KUKA KRL data list: Fadenlegen.dat

&ACCESS RVP
&REL 24
&PARAM DISKPATH = KRC:\R1\myProgramme\Mahlen
DEFDAT  Fadenlegen
;FOLD EXTERNAL DECLARATIONS;%{PE}%MKUKATPBASIS,%CEXT,%VCOMMON,%P
;FOLD BASISTECH EXT;%{PE}%MKUKATPBASIS,%CEXT,%VEXT,%P
EXT  BAS (BAS_COMMAND  :IN,REAL  :IN )
;ENDFOLD (BASISTECH EXT)
;FOLD USER EXT;%{E}%MKUKATPUSER,%CEXT,%VEXT,%P
;Make your modifications here

DECL E6POS KM={X 270.508820,Y 129.418152,Z 50.0000,A 0.0,B -180.000,C 0.0,S 6,T 26,E1 0.0,E2 0.0,E3 0.0,E4 0.0,E5 0.0,E6 0.0}

DECL E6POS test1={X 276.364288,Y 142.737,Z 19.5319443,A 180.000,B -180.000,C 0.0,S 2,T 10,E1 0.0,E2 0.0,E3 0.0,E4 0.0,E5 0.0,E6 0.0}

DECL E6AXIS MyHome={A1 4.82899427,A2 -40.7993927,A3 107.255463,A4 -2.92958689,A5 26.5940895,A6 -79.3028717,E1 0.0,E2 0.0,E3 0.0,E4 0.0,E5 0.0,E6 0.0}

DECL INT turn=1

DECL INT LetztePos
DECL INT len_Punkte=4002; 4002

DECL INT Sturz[180]
Sturz[1]=10
Sturz[2]=10
Sturz[3]=10
Sturz[4]=10
Sturz[5]=10
Sturz[6]=10
Sturz[7]=10
Sturz[8]=10
Sturz[9]=10
Sturz[10]=10
Sturz[11]=10
Sturz[12]=10
Sturz[13]=10
Sturz[14]=10
Sturz[15]=10
Sturz[16]=10
Sturz[17]=10
Sturz[18]=10
Sturz[19]=10
Sturz[20]=10
Sturz[21]=10
Sturz[22]=10
Sturz[23]=10
Sturz[24]=10
Sturz[25]=10
Sturz[26]=10
Sturz[27]=10
Sturz[28]=10
Sturz[29]=10
Sturz[30]=10
Sturz[31]=10
Sturz[32]=10
Sturz[33]=10
Sturz[34]=10
Sturz[35]=10
Sturz[36]=10
Sturz[37]=10
Sturz[38]=10
Sturz[39]=10
Sturz[40]=10
Sturz[41]=10
Sturz[42]=10
Sturz[43]=10
Sturz[44]=10
Sturz[45]=10
Sturz[46]=10
Sturz[47]=10
Sturz[48]=10
Sturz[49]=10
Sturz[50]=10
Sturz[51]=10
Sturz[52]=10
Sturz[53]=10
Sturz[54]=10
Sturz[55]=10
Sturz[56]=10
Sturz[57]=10
Sturz[58]=10
Sturz[59]=10
Sturz[60]=10
Sturz[61]=10
Sturz[62]=10
Sturz[63]=10
Sturz[64]=10
Sturz[65]=10
Sturz[66]=10
Sturz[67]=10
Sturz[68]=10
Sturz[69]=10
Sturz[70]=10
Sturz[71]=10
Sturz[72]=10
Sturz[73]=10
Sturz[74]=10
Sturz[75]=10
Sturz[76]=10
Sturz[77]=10
Sturz[78]=10
Sturz[79]=10
Sturz[80]=10
Sturz[81]=10
Sturz[82]=10
Sturz[83]=10
Sturz[84]=10
Sturz[85]=10
Sturz[86]=10
Sturz[87]=10
Sturz[88]=10
Sturz[89]=10
Sturz[90]=10
Sturz[91]=-10
Sturz[92]=-10
Sturz[93]=-10
Sturz[94]=-10
Sturz[95]=-10
Sturz[96]=-10
Sturz[97]=-10
Sturz[98]=-10
Sturz[99]=-10
Sturz[100]=-10
Sturz[101]=-10
Sturz[102]=-10
Sturz[103]=-10
Sturz[104]=-10
Sturz[105]=-10
Sturz[106]=-10
Sturz[107]=-10
Sturz[108]=-10
Sturz[109]=-10
Sturz[110]=-10
Sturz[111]=-10
Sturz[112]=10
Sturz[113]=10
Sturz[114]=10
Sturz[115]=10
Sturz[116]=10
Sturz[117]=10
Sturz[118]=10
Sturz[119]=10
Sturz[120]=10
Sturz[121]=10
Sturz[122]=10
Sturz[123]=10
Sturz[124]=10
Sturz[125]=10
Sturz[126]=10
Sturz[127]=10
Sturz[128]=10
Sturz[129]=10
Sturz[130]=10
Sturz[131]=10
Sturz[132]=10
Sturz[133]=10
Sturz[134]=10
Sturz[135]=10
Sturz[136]=10
Sturz[137]=10
Sturz[138]=10
Sturz[139]=10
Sturz[140]=10
Sturz[141]=10
Sturz[142]=10
Sturz[143]=10
Sturz[144]=10
Sturz[145]=10
Sturz[146]=10
Sturz[147]=10
Sturz[148]=10
Sturz[149]=10
Sturz[150]=10
Sturz[151]=10
Sturz[152]=10
Sturz[153]=10
Sturz[154]=10
Sturz[155]=10
Sturz[156]=10
Sturz[157]=10
Sturz[158]=10
Sturz[159]=10
Sturz[160]=10
Sturz[161]=10
Sturz[162]=10
Sturz[163]=10
Sturz[164]=10
Sturz[165]=10
Sturz[166]=10
Sturz[167]=10
Sturz[168]=10
Sturz[169]=10
Sturz[170]=10
Sturz[171]=10
Sturz[172]=10
Sturz[173]=10
Sturz[174]=10
Sturz[175]=10
Sturz[176]=10
Sturz[177]=10
Sturz[178]=10
Sturz[179]=10
Sturz[180]=10



DECL INT TEST[374]
TEST[1]=0
TEST[2]=22
TEST[3]=1
TEST[4]=23
TEST[5]=2
TEST[6]=24
TEST[7]=3
TEST[8]=25
TEST[9]=4
TEST[10]=26
TEST[11]=5
TEST[12]=27
TEST[13]=6
TEST[14]=28
TEST[15]=7
TEST[16]=29
TEST[17]=8
TEST[18]=30
TEST[19]=9
TEST[20]=31
TEST[21]=10
TEST[22]=32
TEST[23]=11
TEST[24]=33
TEST[25]=12
TEST[26]=34
TEST[27]=13
TEST[28]=35
TEST[29]=14
TEST[30]=36
TEST[31]=15
TEST[32]=37
TEST[33]=16
TEST[34]=38
TEST[35]=17
TEST[36]=39
TEST[37]=18
TEST[38]=40
TEST[39]=19
TEST[40]=41
TEST[41]=20
TEST[42]=42
TEST[43]=21
TEST[44]=43
TEST[45]=22
TEST[46]=44
TEST[47]=23
TEST[48]=45
TEST[49]=24
TEST[50]=46
TEST[51]=25
TEST[52]=47
TEST[53]=26
TEST[54]=48
TEST[55]=27
TEST[56]=49
TEST[57]=28
TEST[58]=50
TEST[59]=29
TEST[60]=51
TEST[61]=30
TEST[62]=52
TEST[63]=31
TEST[64]=53
TEST[65]=32
TEST[66]=54
TEST[67]=33
TEST[68]=55
TEST[69]=34
TEST[70]=56
TEST[71]=35
TEST[72]=57
TEST[73]=36
TEST[74]=58
TEST[75]=37
TEST[76]=59
TEST[77]=38
TEST[78]=60
TEST[79]=39
TEST[80]=61
TEST[81]=40
TEST[82]=62
TEST[83]=41
TEST[84]=63
TEST[85]=42
TEST[86]=64
TEST[87]=43
TEST[88]=65
TEST[89]=44
TEST[90]=66
TEST[91]=45
TEST[92]=67
TEST[93]=46
TEST[94]=68
TEST[95]=47
TEST[96]=69
TEST[97]=48
TEST[98]=70
TEST[99]=49
TEST[100]=71
TEST[101]=50
TEST[102]=72
TEST[103]=51
TEST[104]=73
TEST[105]=52
TEST[106]=74
TEST[107]=53
TEST[108]=75
TEST[109]=54
TEST[110]=76
TEST[111]=55
TEST[112]=77
TEST[113]=56
TEST[114]=78
TEST[115]=57
TEST[116]=79
TEST[117]=58
TEST[118]=80
TEST[119]=59
TEST[120]=81
TEST[121]=60
TEST[122]=82
TEST[123]=61
TEST[124]=83
TEST[125]=62
TEST[126]=84
TEST[127]=63
TEST[128]=85
TEST[129]=64
TEST[130]=86
TEST[131]=65
TEST[132]=87
TEST[133]=66
TEST[134]=88
TEST[135]=67
TEST[136]=89
TEST[137]=68
TEST[138]=90
TEST[139]=69
TEST[140]=91
TEST[141]=70
TEST[142]=92
TEST[143]=71
TEST[144]=93
TEST[145]=72
TEST[146]=94
TEST[147]=73
TEST[148]=95
TEST[149]=74
TEST[150]=96
TEST[151]=75
TEST[152]=97
TEST[153]=76
TEST[154]=98
TEST[155]=77
TEST[156]=99
TEST[157]=78
TEST[158]=100
TEST[159]=79
TEST[160]=101
TEST[161]=80
TEST[162]=102
TEST[163]=81
TEST[164]=103
TEST[165]=82
TEST[166]=104
TEST[167]=83
TEST[168]=105
TEST[169]=84
TEST[170]=106
TEST[171]=85
TEST[172]=107
TEST[173]=86
TEST[174]=108
TEST[175]=87
TEST[176]=109
TEST[177]=88
TEST[178]=110
TEST[179]=89
TEST[180]=111
TEST[181]=90
TEST[182]=112
TEST[183]=91
TEST[184]=113
TEST[185]=92
TEST[186]=114
TEST[187]=93
TEST[188]=115
TEST[189]=94
TEST[190]=116
TEST[191]=95
TEST[192]=117
TEST[193]=96
TEST[194]=118
TEST[195]=97
TEST[196]=119
TEST[197]=98
TEST[198]=120
TEST[199]=99
TEST[200]=121
TEST[201]=100
TEST[202]=122
TEST[203]=101
TEST[204]=123
TEST[205]=102
TEST[206]=124
TEST[207]=103
TEST[208]=125
TEST[209]=104
TEST[210]=126
TEST[211]=105
TEST[212]=127
TEST[213]=106
TEST[214]=128
TEST[215]=107
TEST[216]=129
TEST[217]=108
TEST[218]=130
TEST[219]=109
TEST[220]=131
TEST[221]=110
TEST[222]=132
TEST[223]=111
TEST[224]=133
TEST[225]=112
TEST[226]=134
TEST[227]=113
TEST[228]=135
TEST[229]=114
TEST[230]=136
TEST[231]=115
TEST[232]=137
TEST[233]=116
TEST[234]=138
TEST[235]=117
TEST[236]=139
TEST[237]=118
TEST[238]=140
TEST[239]=119
TEST[240]=141
TEST[241]=120
TEST[242]=142
TEST[243]=121
TEST[244]=143
TEST[245]=122
TEST[246]=144
TEST[247]=123
TEST[248]=145
TEST[249]=124
TEST[250]=146
TEST[251]=125
TEST[252]=147
TEST[253]=126
TEST[254]=148
TEST[255]=127
TEST[256]=149
TEST[257]=128
TEST[258]=150
TEST[259]=129
TEST[260]=151
TEST[261]=130
TEST[262]=152
TEST[263]=131
TEST[264]=153
TEST[265]=132
TEST[266]=154
TEST[267]=133
TEST[268]=155
TEST[269]=134
TEST[270]=156
TEST[271]=135
TEST[272]=157
TEST[273]=136
TEST[274]=158
TEST[275]=137
TEST[276]=159
TEST[277]=138
TEST[278]=160
TEST[279]=139
TEST[280]=161
TEST[281]=140
TEST[282]=162
TEST[283]=141
TEST[284]=163
TEST[285]=142
TEST[286]=164
TEST[287]=143
TEST[288]=165
TEST[289]=144
TEST[290]=166
TEST[291]=145
TEST[292]=167
TEST[293]=146
TEST[294]=168
TEST[295]=147
TEST[296]=169
TEST[297]=148
TEST[298]=170
TEST[299]=149
TEST[300]=171
TEST[301]=150
TEST[302]=172
TEST[303]=151
TEST[304]=173
TEST[305]=152
TEST[306]=174
TEST[307]=153
TEST[308]=175
TEST[309]=154
TEST[310]=176
TEST[311]=155
TEST[312]=177
TEST[313]=156
TEST[314]=178
TEST[315]=157
TEST[316]=179
TEST[317]=158
TEST[318]=1
TEST[319]=159
TEST[320]=2
TEST[321]=160
TEST[322]=3
TEST[323]=161
TEST[324]=4
TEST[325]=162
TEST[326]=5
TEST[327]=163
TEST[328]=6
TEST[329]=164
TEST[330]=7
TEST[331]=165
TEST[332]=8
TEST[333]=166
TEST[334]=9
TEST[335]=167
TEST[336]=10
TEST[337]=168
TEST[338]=11
TEST[339]=169
TEST[340]=12
TEST[341]=170
TEST[342]=13
TEST[343]=171
TEST[344]=14
TEST[345]=172
TEST[346]=15
TEST[347]=173
TEST[348]=16
TEST[349]=174
TEST[350]=17
TEST[351]=175
TEST[352]=18
TEST[353]=176
TEST[354]=19
TEST[355]=177
TEST[356]=20
TEST[357]=178
TEST[358]=21
TEST[359]=179
TEST[360]=22
TEST[361]=1
TEST[362]=23
TEST[363]=2
TEST[364]=24
TEST[365]=3
TEST[366]=25
TEST[367]=4
TEST[368]=26
TEST[369]=5
TEST[370]=27
TEST[371]=6
TEST[372]=28
TEST[373]=7
TEST[374]=29





DECL INT Punkte[4002]
Punkte[1]=0
Punkte[2]=98
Punkte[3]=1
Punkte[4]=99
Punkte[5]=4
Punkte[6]=76
Punkte[7]=7
Punkte[8]=93
Punkte[9]=169
Punkte[10]=86
Punkte[11]=13
Punkte[12]=123
Punkte[13]=14
Punkte[14]=87
Punkte[15]=170
Punkte[16]=95
Punkte[17]=8
Punkte[18]=77
Punkte[19]=9
Punkte[20]=79
Punkte[21]=161
Punkte[22]=78
Punkte[23]=11
Punkte[24]=109
Punkte[25]=10
Punkte[26]=108
Punkte[27]=43
Punkte[28]=152
Punkte[29]=67
Punkte[30]=144
Punkte[31]=65
Punkte[32]=143
Punkte[33]=64
Punkte[34]=137
Punkte[35]=33
Punkte[36]=99
Punkte[37]=176
Punkte[38]=88
Punkte[39]=163
Punkte[40]=80
Punkte[41]=12
Punkte[42]=81
Punkte[43]=174
Punkte[44]=103
Punkte[45]=5
Punkte[46]=85
Punkte[47]=13
Punkte[48]=112
Punkte[49]=37
Punkte[50]=140
Punkte[51]=58
Punkte[52]=131
Punkte[53]=20
Punkte[54]=120
Punkte[55]=6
Punkte[56]=104
Punkte[57]=179
Punkte[58]=89
Punkte[59]=178
Punkte[60]=75
Punkte[61]=156
Punkte[62]=53
Punkte[63]=168
Punkte[64]=79
Punkte[65]=11
Punkte[66]=78
Punkte[67]=10
Punkte[68]=122
Punkte[69]=9
Punkte[70]=77
Punkte[71]=158
Punkte[72]=84
Punkte[73]=167
Punkte[74]=85
Punkte[75]=4
Punkte[76]=102
Punkte[77]=6
Punkte[78]=91
Punkte[79]=7
Punkte[80]=76
Punkte[81]=157
Punkte[82]=54
Punkte[83]=129
Punkte[84]=53
Punkte[85]=166
Punkte[86]=83
Punkte[87]=165
Punkte[88]=101
Punkte[89]=3
Punkte[90]=98
Punkte[91]=173
Punkte[92]=78
Punkte[93]=160
Punkte[94]=81
Punkte[95]=12
Punkte[96]=80
Punkte[97]=10
Punkte[98]=85
Punkte[99]=168
Punkte[100]=92
Punkte[101]=7
Punkte[102]=121
Punkte[103]=13
Punkte[104]=82
Punkte[105]=148
Punkte[106]=76
Punkte[107]=146
Punkte[108]=75
Punkte[109]=2
Punkte[110]=100
Punkte[111]=4
Punkte[112]=79
Punkte[113]=8
Punkte[114]=106
Punkte[115]=6
Punkte[116]=77
Punkte[117]=9
Punkte[118]=107
Punkte[119]=42
Punkte[120]=151
Punkte[121]=74
Punkte[122]=145
Punkte[123]=73
Punkte[124]=144
Punkte[125]=64
Punkte[126]=143
Punkte[127]=12
Punkte[128]=111
Punkte[129]=36
Punkte[130]=127
Punkte[131]=28
Punkte[132]=126
Punkte[133]=26
Punkte[134]=117
Punkte[135]=14
Punkte[136]=84
Punkte[137]=169
Punkte[138]=87
Punkte[139]=10
Punkte[140]=78
Punkte[141]=159
Punkte[142]=77
Punkte[143]=9
Punkte[144]=79
Punkte[145]=11
Punkte[146]=110
Punkte[147]=8
Punkte[148]=96
Punkte[149]=165
Punkte[150]=101
Punkte[151]=166
Punkte[152]=100
Punkte[153]=36
Punkte[154]=140
Punkte[155]=71
Punkte[156]=154
Punkte[157]=72
Punkte[158]=155
Punkte[159]=52
Punkte[160]=167
Punkte[161]=91
Punkte[162]=17
Punkte[163]=124
Punkte[164]=15
Punkte[165]=123
Punkte[166]=12
Punkte[167]=82
Punkte[168]=177
Punkte[169]=80
Punkte[170]=162
Punkte[171]=84
Punkte[172]=3
Punkte[173]=76
Punkte[174]=157
Punkte[175]=77
Punkte[176]=8
Punkte[177]=78
Punkte[178]=164
Punkte[179]=81
Punkte[180]=174
Punkte[181]=87
Punkte[182]=163
Punkte[183]=49
Punkte[184]=119
Punkte[185]=19
Punkte[186]=124
Punkte[187]=16
Punkte[188]=90
Punkte[189]=179
Punkte[190]=73
Punkte[191]=1
Punkte[192]=79
Punkte[193]=10
Punkte[194]=86
Punkte[195]=14
Punkte[196]=111
Punkte[197]=11
Punkte[198]=77
Punkte[199]=146
Punkte[200]=74
Punkte[201]=118
Punkte[202]=48
Punkte[203]=162
Punkte[204]=82
Punkte[205]=148
Punkte[206]=83
Punkte[207]=3
Punkte[208]=99
Punkte[209]=9
Punkte[210]=80
Punkte[211]=12
Punkte[212]=81
Punkte[213]=175
Punkte[214]=98
Punkte[215]=170
Punkte[216]=102
Punkte[217]=168
Punkte[218]=84
Punkte[219]=5
Punkte[220]=75
Punkte[221]=6
Punkte[222]=79
Punkte[223]=147
Punkte[224]=74
Punkte[225]=1
Punkte[226]=94
Punkte[227]=169
Punkte[228]=56
Punkte[229]=139
Punkte[230]=70
Punkte[231]=153
Punkte[232]=78
Punkte[233]=11
Punkte[234]=105
Punkte[235]=3
Punkte[236]=97
Punkte[237]=172
Punkte[238]=96
Punkte[239]=2
Punkte[240]=103
Punkte[241]=39
Punkte[242]=104
Punkte[243]=178
Punkte[244]=72
Punkte[245]=177
Punkte[246]=102
Punkte[247]=171
Punkte[248]=80
Punkte[249]=147
Punkte[250]=75
Punkte[251]=155
Punkte[252]=74
Punkte[253]=118
Punkte[254]=11
Punkte[255]=77
Punkte[256]=10
Punkte[257]=81
Punkte[258]=163
Punkte[259]=93
Punkte[260]=7
Punkte[261]=78
Punkte[262]=12
Punkte[263]=110
Punkte[264]=35
Punkte[265]=100
Punkte[266]=36
Punkte[267]=102
Punkte[268]=5
Punkte[269]=101
Punkte[270]=4
Punkte[271]=112
Punkte[272]=13
Punkte[273]=120
Punkte[274]=21
Punkte[275]=122
Punkte[276]=11
Punkte[277]=109
Punkte[278]=34
Punkte[279]=139
Punkte[280]=87
Punkte[281]=15
Punkte[282]=124
Punkte[283]=14
Punkte[284]=123
Punkte[285]=12
Punkte[286]=142
Punkte[287]=72
Punkte[288]=144
Punkte[289]=66
Punkte[290]=131
Punkte[291]=20
Punkte[292]=97
Punkte[293]=165
Punkte[294]=101
Punkte[295]=166
Punkte[296]=82
Punkte[297]=13
Punkte[298]=85
Punkte[299]=159
Punkte[300]=46
Punkte[301]=115
Punkte[302]=10
Punkte[303]=122
Punkte[304]=9
Punkte[305]=77
Punkte[306]=127
Punkte[307]=36
Punkte[308]=111
Punkte[309]=12
Punkte[310]=116
Punkte[311]=11
Punkte[312]=80
Punkte[313]=4
Punkte[314]=86
Punkte[315]=173
Punkte[316]=96
Punkte[317]=8
Punkte[318]=79
Punkte[319]=3
Punkte[320]=108
Punkte[321]=2
Punkte[322]=84
Punkte[323]=166
Punkte[324]=83
Punkte[325]=5
Punkte[326]=77
Punkte[327]=7
Punkte[328]=76
Punkte[329]=149
Punkte[330]=85
Punkte[331]=160
Punkte[332]=89
Punkte[333]=179
Punkte[334]=75
Punkte[335]=146
Punkte[336]=82
Punkte[337]=11
Punkte[338]=104
Punkte[339]=172
Punkte[340]=98
Punkte[341]=29
Punkte[342]=126
Punkte[343]=17
Punkte[344]=152
Punkte[345]=16
Punkte[346]=125
Punkte[347]=23
Punkte[348]=123
Punkte[349]=13
Punkte[350]=84
Punkte[351]=12
Punkte[352]=80
Punkte[353]=174
Punkte[354]=81
Punkte[355]=175
Punkte[356]=100
Punkte[357]=168
Punkte[358]=53
Punkte[359]=156
Punkte[360]=77
Punkte[361]=8
Punkte[362]=95
Punkte[363]=169
Punkte[364]=85
Punkte[365]=171
Punkte[366]=101
Punkte[367]=167
Punkte[368]=83
Punkte[369]=4
Punkte[370]=99
Punkte[371]=32
Punkte[372]=138
Punkte[373]=69
Punkte[374]=153
Punkte[375]=18
Punkte[376]=124
Punkte[377]=13
Punkte[378]=111
Punkte[379]=45
Punkte[380]=158
Punkte[381]=78
Punkte[382]=12
Punkte[383]=81
Punkte[384]=11
Punkte[385]=77
Punkte[386]=127
Punkte[387]=17
Punkte[388]=125
Punkte[389]=24
Punkte[390]=116
Punkte[391]=47
Punkte[392]=161
Punkte[393]=79
Punkte[394]=7
Punkte[395]=102
Punkte[396]=167
Punkte[397]=86
Punkte[398]=6
Punkte[399]=121
Punkte[400]=8
Punkte[401]=84
Punkte[402]=10
Punkte[403]=136
Punkte[404]=50
Punkte[405]=165
Punkte[406]=78
Punkte[407]=176
Punkte[408]=77
Punkte[409]=128
Punkte[410]=0
Punkte[411]=93
Punkte[412]=164
Punkte[413]=82
Punkte[414]=148
Punkte[415]=14
Punkte[416]=87
Punkte[417]=150
Punkte[418]=15
Punkte[419]=151
Punkte[420]=89
Punkte[421]=178
Punkte[422]=103
Punkte[423]=10
Punkte[424]=88
Punkte[425]=141
Punkte[426]=60
Punkte[427]=170
Punkte[428]=94
Punkte[429]=7
Punkte[430]=121
Punkte[431]=75
Punkte[432]=3
Punkte[433]=101
Punkte[434]=11
Punkte[435]=78
Punkte[436]=172
Punkte[437]=80
Punkte[438]=12
Punkte[439]=79
Punkte[440]=5
Punkte[441]=76
Punkte[442]=157
Punkte[443]=54
Punkte[444]=168
Punkte[445]=97
Punkte[446]=2
Punkte[447]=132
Punkte[448]=29
Punkte[449]=127
Punkte[450]=77
Punkte[451]=161
Punkte[452]=91
Punkte[453]=7
Punkte[454]=105
Punkte[455]=167
Punkte[456]=99
Punkte[457]=33
Punkte[458]=101
Punkte[459]=165
Punkte[460]=51
Punkte[461]=154
Punkte[462]=44
Punkte[463]=109
Punkte[464]=4
Punkte[465]=84
Punkte[466]=159
Punkte[467]=86
Punkte[468]=169
Punkte[469]=57
Punkte[470]=160
Punkte[471]=78
Punkte[472]=10
Punkte[473]=82
Punkte[474]=12
Punkte[475]=142
Punkte[476]=55
Punkte[477]=158
Punkte[478]=83
Punkte[479]=11
Punkte[480]=92
Punkte[481]=0
Punkte[482]=128
Punkte[483]=38
Punkte[484]=103
Punkte[485]=174
Punkte[486]=81
Punkte[487]=157
Punkte[488]=47
Punkte[489]=164
Punkte[490]=99
Punkte[491]=175
Punkte[492]=91
Punkte[493]=6
Punkte[494]=76
Punkte[495]=7
Punkte[496]=84
Punkte[497]=134
Punkte[498]=85
Punkte[499]=140
Punkte[500]=52
Punkte[501]=155
Punkte[502]=45
Punkte[503]=158
Punkte[504]=48
Punkte[505]=118
Punkte[506]=74
Punkte[507]=145
Punkte[508]=75
Punkte[509]=156
Punkte[510]=53
Punkte[511]=166
Punkte[512]=90
Punkte[513]=0
Punkte[514]=128
Punkte[515]=18
Punkte[516]=125
Punkte[517]=25
Punkte[518]=126
Punkte[519]=31
Punkte[520]=133
Punkte[521]=79
Punkte[522]=11
Punkte[523]=119
Punkte[524]=12
Punkte[525]=78
Punkte[526]=168
Punkte[527]=60
Punkte[528]=170
Punkte[529]=59
Punkte[530]=141
Punkte[531]=88
Punkte[532]=150
Punkte[533]=15
Punkte[534]=151
Punkte[535]=16
Punkte[536]=91
Punkte[537]=166
Punkte[538]=101
Punkte[539]=37
Punkte[540]=112
Punkte[541]=13
Punkte[542]=123
Punkte[543]=14
Punkte[544]=93
Punkte[545]=171
Punkte[546]=62
Punkte[547]=142
Punkte[548]=63
Punkte[549]=143
Punkte[550]=12
Punkte[551]=83
Punkte[552]=165
Punkte[553]=96
Punkte[554]=164
Punkte[555]=88
Punkte[556]=140
Punkte[557]=52
Punkte[558]=166
Punkte[559]=102
Punkte[560]=37
Punkte[561]=112
Punkte[562]=177
Punkte[563]=94
Punkte[564]=0
Punkte[565]=128
Punkte[566]=179
Punkte[567]=77
Punkte[568]=153
Punkte[569]=70
Punkte[570]=145
Punkte[571]=69
Punkte[572]=171
Punkte[573]=98
Punkte[574]=1
Punkte[575]=130
Punkte[576]=55
Punkte[577]=169
Punkte[578]=56
Punkte[579]=159
Punkte[580]=85
Punkte[581]=170
Punkte[582]=89
Punkte[583]=142
Punkte[584]=61
Punkte[585]=137
Punkte[586]=52
Punkte[587]=165
Punkte[588]=100
Punkte[589]=36
Punkte[590]=139
Punkte[591]=50
Punkte[592]=164
Punkte[593]=92
Punkte[594]=10
Punkte[595]=136
Punkte[596]=11
Punkte[597]=77
Punkte[598]=8
Punkte[599]=91
Punkte[600]=179
Punkte[601]=90
Punkte[602]=6
Punkte[603]=87
Punkte[604]=170
Punkte[605]=103
Punkte[606]=177
Punkte[607]=82
Punkte[608]=3
Punkte[609]=76
Punkte[610]=125
Punkte[611]=15
Punkte[612]=88
Punkte[613]=141
Punkte[614]=12
Punkte[615]=81
Punkte[616]=133
Punkte[617]=78
Punkte[618]=9
Punkte[619]=108
Punkte[620]=43
Punkte[621]=156
Punkte[622]=84
Punkte[623]=157
Punkte[624]=54
Punkte[625]=138
Punkte[626]=70
Punkte[627]=115
Punkte[628]=46
Punkte[629]=112
Punkte[630]=16
Punkte[631]=113
Punkte[632]=6
Punkte[633]=105
Punkte[634]=172
Punkte[635]=95
Punkte[636]=11
Punkte[637]=106
Punkte[638]=41
Punkte[639]=149
Punkte[640]=77
Punkte[641]=10
Punkte[642]=122
Punkte[643]=14
Punkte[644]=84
Punkte[645]=158
Punkte[646]=76
Punkte[647]=146
Punkte[648]=75
Punkte[649]=5
Punkte[650]=135
Punkte[651]=7
Punkte[652]=93
Punkte[653]=176
Punkte[654]=102
Punkte[655]=168
Punkte[656]=55
Punkte[657]=142
Punkte[658]=66
Punkte[659]=172
Punkte[660]=96
Punkte[661]=154
Punkte[662]=71
Punkte[663]=116
Punkte[664]=72
Punkte[665]=145
Punkte[666]=74
Punkte[667]=119
Punkte[668]=151
Punkte[669]=65
Punkte[670]=144
Punkte[671]=64
Punkte[672]=166
Punkte[673]=99
Punkte[674]=174
Punkte[675]=91
Punkte[676]=10
Punkte[677]=83
Punkte[678]=179
Punkte[679]=118
Punkte[680]=150
Punkte[681]=77
Punkte[682]=9
Punkte[683]=79
Punkte[684]=167
Punkte[685]=56
Punkte[686]=131
Punkte[687]=19
Punkte[688]=95
Punkte[689]=2
Punkte[690]=76
Punkte[691]=149
Punkte[692]=69
Punkte[693]=138
Punkte[694]=87
Punkte[695]=4
Punkte[696]=129
Punkte[697]=0
Punkte[698]=74
Punkte[699]=3
Punkte[700]=107
Punkte[701]=8
Punkte[702]=128
Punkte[703]=30
Punkte[704]=126
Punkte[705]=26
Punkte[706]=97
Punkte[707]=1
Punkte[708]=130
Punkte[709]=12
Punkte[710]=92
Punkte[711]=167
Punkte[712]=84
Punkte[713]=6
Punkte[714]=85
Punkte[715]=5
Punkte[716]=116
Punkte[717]=172
Punkte[718]=86
Punkte[719]=13
Punkte[720]=78
Punkte[721]=10
Punkte[722]=136
Punkte[723]=63
Punkte[724]=171
Punkte[725]=74
Punkte[726]=118
Punkte[727]=28
Punkte[728]=127
Punkte[729]=36
Punkte[730]=102
Punkte[731]=169
Punkte[732]=87
Punkte[733]=175
Punkte[734]=88
Punkte[735]=140
Punkte[736]=38
Punkte[737]=114
Punkte[738]=45
Punkte[739]=162
Punkte[740]=92
Punkte[741]=161
Punkte[742]=47
Punkte[743]=113
Punkte[744]=14
Punkte[745]=137
Punkte[746]=86
Punkte[747]=15
Punkte[748]=89
Punkte[749]=151
Punkte[750]=42
Punkte[751]=104
Punkte[752]=167
Punkte[753]=102
Punkte[754]=10
Punkte[755]=108
Punkte[756]=33
Punkte[757]=99
Punkte[758]=160
Punkte[759]=56
Punkte[760]=169
Punkte[761]=101
Punkte[762]=2
Punkte[763]=77
Punkte[764]=3
Punkte[765]=133
Punkte[766]=79
Punkte[767]=11
Punkte[768]=78
Punkte[769]=163
Punkte[770]=89
Punkte[771]=165
Punkte[772]=98
Punkte[773]=9
Punkte[774]=100
Punkte[775]=4
Punkte[776]=85
Punkte[777]=140
Punkte[778]=36
Punkte[779]=111
Punkte[780]=12
Punkte[781]=120
Punkte[782]=13
Punkte[783]=143
Punkte[784]=58
Punkte[785]=161
Punkte[786]=75
Punkte[787]=1
Punkte[788]=84
Punkte[789]=3
Punkte[790]=128
Punkte[791]=77
Punkte[792]=158
Punkte[793]=31
Punkte[794]=139
Punkte[795]=35
Punkte[796]=110
Punkte[797]=8
Punkte[798]=106
Punkte[799]=44
Punkte[800]=157
Punkte[801]=78
Punkte[802]=12
Punkte[803]=115
Punkte[804]=39
Punkte[805]=103
Punkte[806]=5
Punkte[807]=88
Punkte[808]=141
Punkte[809]=53
Punkte[810]=168
Punkte[811]=101
Punkte[812]=171
Punkte[813]=92
Punkte[814]=17
Punkte[815]=152
Punkte[816]=120
Punkte[817]=4
Punkte[818]=111
Punkte[819]=11
Punkte[820]=130
Punkte[821]=57
Punkte[822]=110
Punkte[823]=13
Punkte[824]=82
Punkte[825]=156
Punkte[826]=46
Punkte[827]=115
Punkte[828]=69
Punkte[829]=139
Punkte[830]=70
Punkte[831]=150
Punkte[832]=88
Punkte[833]=12
Punkte[834]=136
Punkte[835]=85
Punkte[836]=10
Punkte[837]=86
Punkte[838]=166
Punkte[839]=53
Punkte[840]=141
Punkte[841]=71
Punkte[842]=176
Punkte[843]=101
Punkte[844]=167
Punkte[845]=78
Punkte[846]=156
Punkte[847]=74
Punkte[848]=179
Punkte[849]=89
Punkte[850]=164
Punkte[851]=100
Punkte[852]=3
Punkte[853]=83
Punkte[854]=178
Punkte[855]=102
Punkte[856]=2
Punkte[857]=132
Punkte[858]=26
Punkte[859]=155
Punkte[860]=79
Punkte[861]=134
Punkte[862]=4
Punkte[863]=76
Punkte[864]=145
Punkte[865]=71
Punkte[866]=140
Punkte[867]=58
Punkte[868]=130
Punkte[869]=56
Punkte[870]=139
Punkte[871]=11
Punkte[872]=77
Punkte[873]=163
Punkte[874]=80
Punkte[875]=10
Punkte[876]=122
Punkte[877]=24
Punkte[878]=138
Punkte[879]=67
Punkte[880]=144
Punkte[881]=13
Punkte[882]=89
Punkte[883]=141
Punkte[884]=61
Punkte[885]=112
Punkte[886]=170
Punkte[887]=90
Punkte[888]=135
Punkte[889]=79
Punkte[890]=154
Punkte[891]=71
Punkte[892]=175
Punkte[893]=83
Punkte[894]=2
Punkte[895]=78
Punkte[896]=159
Punkte[897]=34
Punkte[898]=100
Punkte[899]=7
Punkte[900]=121
Punkte[901]=6
Punkte[902]=129
Punkte[903]=4
Punkte[904]=74
Punkte[905]=146
Punkte[906]=82
Punkte[907]=134
Punkte[908]=85
Punkte[909]=149
Punkte[910]=86
Punkte[911]=168
Punkte[912]=59
Punkte[913]=171
Punkte[914]=62
Punkte[915]=150
Punkte[916]=79
Punkte[917]=9
Punkte[918]=84
Punkte[919]=140
Punkte[920]=52
Punkte[921]=155
Punkte[922]=73
Punkte[923]=117
Punkte[924]=173
Punkte[925]=100
Punkte[926]=166
Punkte[927]=101
Punkte[928]=165
Punkte[929]=90
Punkte[930]=10
Punkte[931]=95
Punkte[932]=178
Punkte[933]=89
Punkte[934]=16
Punkte[935]=126
Punkte[936]=76
Punkte[937]=149
Punkte[938]=14
Punkte[939]=83
Punkte[940]=148
Punkte[941]=82
Punkte[942]=175
Punkte[943]=74
Punkte[944]=144
Punkte[945]=65
Punkte[946]=137
Punkte[947]=63
Punkte[948]=141
Punkte[949]=87
Punkte[950]=138
Punkte[951]=34
Punkte[952]=109
Punkte[953]=11
Punkte[954]=105
Punkte[955]=40
Punkte[956]=129
Punkte[957]=8
Punkte[958]=78
Punkte[959]=164
Punkte[960]=99
Punkte[961]=32
Punkte[962]=158
Punkte[963]=55
Punkte[964]=130
Punkte[965]=19
Punkte[966]=126
Punkte[967]=27
Punkte[968]=127
Punkte[969]=174
Punkte[970]=110
Punkte[971]=44
Punkte[972]=156
Punkte[973]=53
Punkte[974]=108
Punkte[975]=3
Punkte[976]=98
Punkte[977]=30
Punkte[978]=139
Punkte[979]=33
Punkte[980]=159
Punkte[981]=79
Punkte[982]=4
Punkte[983]=135
Punkte[984]=10
Punkte[985]=81
Punkte[986]=11
Punkte[987]=123
Punkte[988]=13
Punkte[989]=78
Punkte[990]=7
Punkte[991]=86
Punkte[992]=5
Punkte[993]=129
Punkte[994]=0
Punkte[995]=73
Punkte[996]=117
Punkte[997]=26
Punkte[998]=154
Punkte[999]=93
Punkte[1000]=18
Punkte[1001]=153
Punkte[1002]=51
Punkte[1003]=164
Punkte[1004]=48
Punkte[1005]=138
Punkte[1006]=54
Punkte[1007]=166
Punkte[1008]=83
Punkte[1009]=140
Punkte[1010]=88
Punkte[1011]=179
Punkte[1012]=127
Punkte[1013]=35
Punkte[1014]=100
Punkte[1015]=11
Punkte[1016]=78
Punkte[1017]=10
Punkte[1018]=89
Punkte[1019]=173
Punkte[1020]=97
Punkte[1021]=15
Punkte[1022]=151
Punkte[1023]=119
Punkte[1024]=174
Punkte[1025]=72
Punkte[1026]=177
Punkte[1027]=73
Punkte[1028]=143
Punkte[1029]=62
Punkte[1030]=140
Punkte[1031]=85
Punkte[1032]=12
Punkte[1033]=80
Punkte[1034]=165
Punkte[1035]=99
Punkte[1036]=160
Punkte[1037]=74
Punkte[1038]=125
Punkte[1039]=76
Punkte[1040]=179
Punkte[1041]=104
Punkte[1042]=172
Punkte[1043]=105
Punkte[1044]=167
Punkte[1045]=87
Punkte[1046]=13
Punkte[1047]=142
Punkte[1048]=89
Punkte[1049]=143
Punkte[1050]=66
Punkte[1051]=144
Punkte[1052]=72
Punkte[1053]=155
Punkte[1054]=75
Punkte[1055]=145
Punkte[1056]=14
Punkte[1057]=124
Punkte[1058]=15
Punkte[1059]=123
Punkte[1060]=178
Punkte[1061]=88
Punkte[1062]=174
Punkte[1063]=127
Punkte[1064]=30
Punkte[1065]=100
Punkte[1066]=36
Punkte[1067]=160
Punkte[1068]=19
Punkte[1069]=119
Punkte[1070]=74
Punkte[1071]=126
Punkte[1072]=29
Punkte[1073]=98
Punkte[1074]=0
Punkte[1075]=77
Punkte[1076]=162
Punkte[1077]=93
Punkte[1078]=10
Punkte[1079]=140
Punkte[1080]=37
Punkte[1081]=102
Punkte[1082]=8
Punkte[1083]=94
Punkte[1084]=17
Punkte[1085]=152
Punkte[1086]=43
Punkte[1087]=111
Punkte[1088]=4
Punkte[1089]=99
Punkte[1090]=3
Punkte[1091]=128
Punkte[1092]=31
Punkte[1093]=132
Punkte[1094]=72
Punkte[1095]=117
Punkte[1096]=11
Punkte[1097]=86
Punkte[1098]=159
Punkte[1099]=77
Punkte[1100]=151
Punkte[1101]=16
Punkte[1102]=124
Punkte[1103]=75
Punkte[1104]=120
Punkte[1105]=153
Punkte[1106]=23
Punkte[1107]=125
Punkte[1108]=24
Punkte[1109]=116
Punkte[1110]=12
Punkte[1111]=114
Punkte[1112]=68
Punkte[1113]=9
Punkte[1114]=80
Punkte[1115]=170
Punkte[1116]=97
Punkte[1117]=20
Punkte[1118]=131
Punkte[1119]=2
Punkte[1120]=82
Punkte[1121]=178
Punkte[1122]=134
Punkte[1123]=77
Punkte[1124]=8
Punkte[1125]=96
Punkte[1126]=154
Punkte[1127]=73
Punkte[1128]=172
Punkte[1129]=72
Punkte[1130]=176
Punkte[1131]=92
Punkte[1132]=151
Punkte[1133]=78
Punkte[1134]=4
Punkte[1135]=130
Punkte[1136]=54
Punkte[1137]=157
Punkte[1138]=84
Punkte[1139]=11
Punkte[1140]=79
Punkte[1141]=129
Punkte[1142]=19
Punkte[1143]=97
Punkte[1144]=169
Punkte[1145]=57
Punkte[1146]=143
Punkte[1147]=63
Punkte[1148]=171
Punkte[1149]=102
Punkte[1150]=166
Punkte[1151]=98
Punkte[1152]=32
Punkte[1153]=99
Punkte[1154]=168
Punkte[1155]=60
Punkte[1156]=135
Punkte[1157]=90
Punkte[1158]=174
Punkte[1159]=96
Punkte[1160]=11
Punkte[1161]=89
Punkte[1162]=12
Punkte[1163]=82
Punkte[1164]=147
Punkte[1165]=80
Punkte[1166]=133
Punkte[1167]=81
Punkte[1168]=3
Punkte[1169]=106
Punkte[1170]=177
Punkte[1171]=112
Punkte[1172]=13
Punkte[1173]=136
Punkte[1174]=9
Punkte[1175]=72
Punkte[1176]=113
Punkte[1177]=44
Punkte[1178]=109
Punkte[1179]=55
Punkte[1180]=169
Punkte[1181]=94
Punkte[1182]=165
Punkte[1183]=91
Punkte[1184]=7
Punkte[1185]=92
Punkte[1186]=18
Punkte[1187]=158
Punkte[1188]=84
Punkte[1189]=14
Punkte[1190]=148
Punkte[1191]=40
Punkte[1192]=115
Punkte[1193]=70
Punkte[1194]=171
Punkte[1195]=100
Punkte[1196]=162
Punkte[1197]=78
Punkte[1198]=173
Punkte[1199]=88
Punkte[1200]=163
Punkte[1201]=97
Punkte[1202]=172
Punkte[1203]=77
Punkte[1204]=10
Punkte[1205]=75
Punkte[1206]=126
Punkte[1207]=23
Punkte[1208]=80
Punkte[1209]=11
Punkte[1210]=85
Punkte[1211]=141
Punkte[1212]=64
Punkte[1213]=142
Punkte[1214]=93
Punkte[1215]=1
Punkte[1216]=128
Punkte[1217]=179
Punkte[1218]=118
Punkte[1219]=150
Punkte[1220]=16
Punkte[1221]=152
Punkte[1222]=120
Punkte[1223]=6
Punkte[1224]=117
Punkte[1225]=176
Punkte[1226]=78
Punkte[1227]=130
Punkte[1228]=42
Punkte[1229]=155
Punkte[1230]=27
Punkte[1231]=97
Punkte[1232]=167
Punkte[1233]=104
Punkte[1234]=12
Punkte[1235]=110
Punkte[1236]=11
Punkte[1237]=103
Punkte[1238]=169
Punkte[1239]=84
Punkte[1240]=5
Punkte[1241]=101
Punkte[1242]=3
Punkte[1243]=73
Punkte[1244]=1
Punkte[1245]=74
Punkte[1246]=178
Punkte[1247]=124
Punkte[1248]=76
Punkte[1249]=8
Punkte[1250]=105
Punkte[1251]=10
Punkte[1252]=130
Punkte[1253]=59
Punkte[1254]=137
Punkte[1255]=61
Punkte[1256]=146
Punkte[1257]=77
Punkte[1258]=7
Punkte[1259]=107
Punkte[1260]=2
Punkte[1261]=108
Punkte[1262]=9
Punkte[1263]=85
Punkte[1264]=15
Punkte[1265]=87
Punkte[1266]=176
Punkte[1267]=88
Punkte[1268]=14
Punkte[1269]=123
Punkte[1270]=12
Punkte[1271]=118
Punkte[1272]=150
Punkte[1273]=89
Punkte[1274]=172
Punkte[1275]=109
Punkte[1276]=70
Punkte[1277]=138
Punkte[1278]=67
Punkte[1279]=135
Punkte[1280]=5
Punkte[1281]=132
Punkte[1282]=21
Punkte[1283]=98
Punkte[1284]=1
Punkte[1285]=78
Punkte[1286]=153
Punkte[1287]=77
Punkte[1288]=6
Punkte[1289]=103
Punkte[1290]=166
Punkte[1291]=52
Punkte[1292]=142
Punkte[1293]=12
Punkte[1294]=81
Punkte[1295]=175
Punkte[1296]=101
Punkte[1297]=33
Punkte[1298]=134
Punkte[1299]=178
Punkte[1300]=73
Punkte[1301]=160
Punkte[1302]=85
Punkte[1303]=3
Punkte[1304]=97
Punkte[1305]=156
Punkte[1306]=75
Punkte[1307]=132
Punkte[1308]=28
Punkte[1309]=135
Punkte[1310]=90
Punkte[1311]=151
Punkte[1312]=65
Punkte[1313]=143
Punkte[1314]=59
Punkte[1315]=170
Punkte[1316]=57
Punkte[1317]=161
Punkte[1318]=95
Punkte[1319]=173
Punkte[1320]=99
Punkte[1321]=34
Punkte[1322]=139
Punkte[1323]=50
Punkte[1324]=165
Punkte[1325]=96
Punkte[1326]=23
Punkte[1327]=98
Punkte[1328]=179
Punkte[1329]=126
Punkte[1330]=174
Punkte[1331]=102
Punkte[1332]=168
Punkte[1333]=106
Punkte[1334]=25
Punkte[1335]=156
Punkte[1336]=76
Punkte[1337]=144
Punkte[1338]=73
Punkte[1339]=145
Punkte[1340]=13
Punkte[1341]=78
Punkte[1342]=3
Punkte[1343]=104
Punkte[1344]=40
Punkte[1345]=117
Punkte[1346]=42
Punkte[1347]=110
Punkte[1348]=4
Punkte[1349]=112
Punkte[1350]=12
Punkte[1351]=86
Punkte[1352]=137
Punkte[1353]=16
Punkte[1354]=88
Punkte[1355]=177
Punkte[1356]=113
Punkte[1357]=171
Punkte[1358]=80
Punkte[1359]=138
Punkte[1360]=61
Punkte[1361]=111
Punkte[1362]=45
Punkte[1363]=106
Punkte[1364]=179
Punkte[1365]=103
Punkte[1366]=175
Punkte[1367]=92
Punkte[1368]=20
Punkte[1369]=114
Punkte[1370]=38
Punkte[1371]=131
Punkte[1372]=63
Punkte[1373]=136
Punkte[1374]=85
Punkte[1375]=13
Punkte[1376]=130
Punkte[1377]=1
Punkte[1378]=72
Punkte[1379]=9
Punkte[1380]=99
Punkte[1381]=164
Punkte[1382]=79
Punkte[1383]=8
Punkte[1384]=87
Punkte[1385]=10
Punkte[1386]=74
Punkte[1387]=124
Punkte[1388]=7
Punkte[1389]=76
Punkte[1390]=5
Punkte[1391]=75
Punkte[1392]=133
Punkte[1393]=22
Punkte[1394]=104
Punkte[1395]=172
Punkte[1396]=69
Punkte[1397]=171
Punkte[1398]=78
Punkte[1399]=154
Punkte[1400]=21
Punkte[1401]=115
Punkte[1402]=175
Punkte[1403]=121
Punkte[1404]=153
Punkte[1405]=92
Punkte[1406]=12
Punkte[1407]=119
Punkte[1408]=49
Punkte[1409]=163
Punkte[1410]=76
Punkte[1411]=152
Punkte[1412]=120
Punkte[1413]=11
Punkte[1414]=102
Punkte[1415]=167
Punkte[1416]=94
Punkte[1417]=166
Punkte[1418]=66
Punkte[1419]=170
Punkte[1420]=82
Punkte[1421]=134
Punkte[1422]=6
Punkte[1423]=91
Punkte[1424]=148
Punkte[1425]=88
Punkte[1426]=15
Punkte[1427]=79
Punkte[1428]=10
Punkte[1429]=114
Punkte[1430]=64
Punkte[1431]=151
Punkte[1432]=42
Punkte[1433]=120
Punkte[1434]=74
Punkte[1435]=177
Punkte[1436]=81
Punkte[1437]=11
Punkte[1438]=113
Punkte[1439]=65
Punkte[1440]=138
Punkte[1441]=33
Punkte[1442]=99
Punkte[1443]=26
Punkte[1444]=126
Punkte[1445]=24
Punkte[1446]=127
Punkte[1447]=37
Punkte[1448]=101
Punkte[1449]=170
Punkte[1450]=102
Punkte[1451]=7
Punkte[1452]=129
Punkte[1453]=4
Punkte[1454]=85
Punkte[1455]=168
Punkte[1456]=90
Punkte[1457]=0
Punkte[1458]=76
Punkte[1459]=146
Punkte[1460]=82
Punkte[1461]=165
Punkte[1462]=77
Punkte[1463]=1
Punkte[1464]=92
Punkte[1465]=152
Punkte[1466]=67
Punkte[1467]=103
Punkte[1468]=174
Punkte[1469]=127
Punkte[1470]=31
Punkte[1471]=126
Punkte[1472]=2
Punkte[1473]=75
Punkte[1474]=139
Punkte[1475]=70
Punkte[1476]=108
Punkte[1477]=168
Punkte[1478]=55
Punkte[1479]=158
Punkte[1480]=18
Punkte[1481]=119
Punkte[1482]=10
Punkte[1483]=86
Punkte[1484]=143
Punkte[1485]=58
Punkte[1486]=169
Punkte[1487]=93
Punkte[1488]=149
Punkte[1489]=117
Punkte[1490]=150
Punkte[1491]=66
Punkte[1492]=172
Punkte[1493]=76
Punkte[1494]=4
Punkte[1495]=135
Punkte[1496]=3
Punkte[1497]=134
Punkte[1498]=84
Punkte[1499]=140
Punkte[1500]=59
Punkte[1501]=141
Punkte[1502]=44
Punkte[1503]=131
Punkte[1504]=51
Punkte[1505]=161
Punkte[1506]=91
Punkte[1507]=15
Punkte[1508]=112
Punkte[1509]=64
Punkte[1510]=144
Punkte[1511]=14
Punkte[1512]=125
Punkte[1513]=17
Punkte[1514]=124
Punkte[1515]=29
Punkte[1516]=126
Punkte[1517]=77
Punkte[1518]=139
Punkte[1519]=68
Punkte[1520]=9
Punkte[1521]=73
Punkte[1522]=132
Punkte[1523]=57
Punkte[1524]=167
Punkte[1525]=56
Punkte[1526]=143
Punkte[1527]=70
Punkte[1528]=173
Punkte[1529]=87
Punkte[1530]=168
Punkte[1531]=105
Punkte[1532]=13
Punkte[1533]=146
Punkte[1534]=15
Punkte[1535]=149
Punkte[1536]=116
Punkte[1537]=71
Punkte[1538]=174
Punkte[1539]=104
Punkte[1540]=177
Punkte[1541]=82
Punkte[1542]=0
Punkte[1543]=92
Punkte[1544]=19
Punkte[1545]=160
Punkte[1546]=95
Punkte[1547]=152
Punkte[1548]=43
Punkte[1549]=112
Punkte[1550]=170
Punkte[1551]=87
Punkte[1552]=164
Punkte[1553]=96
Punkte[1554]=179
Punkte[1555]=90
Punkte[1556]=14
Punkte[1557]=86
Punkte[1558]=13
Punkte[1559]=97
Punkte[1560]=20
Punkte[1561]=154
Punkte[1562]=121
Punkte[1563]=155
Punkte[1564]=77
Punkte[1565]=143
Punkte[1566]=76
Punkte[1567]=1
Punkte[1568]=123
Punkte[1569]=28
Punkte[1570]=157
Punkte[1571]=78
Punkte[1572]=12
Punkte[1573]=79
Punkte[1574]=165
Punkte[1575]=83
Punkte[1576]=11
Punkte[1577]=101
Punkte[1578]=38
Punkte[1579]=140
Punkte[1580]=39
Punkte[1581]=148
Punkte[1582]=48
Punkte[1583]=118
Punkte[1584]=73
Punkte[1585]=153
Punkte[1586]=16
Punkte[1587]=97
Punkte[1588]=175
Punkte[1589]=82
Punkte[1590]=3
Punkte[1591]=76
Punkte[1592]=127
Punkte[1593]=25
Punkte[1594]=128
Punkte[1595]=27
Punkte[1596]=122
Punkte[1597]=11
Punkte[1598]=105
Punkte[1599]=172
Punkte[1600]=115
Punkte[1601]=22
Punkte[1602]=98
Punkte[1603]=165
Punkte[1604]=93
Punkte[1605]=171
Punkte[1606]=94
Punkte[1607]=142
Punkte[1608]=15
Punkte[1609]=137
Punkte[1610]=57
Punkte[1611]=130
Punkte[1612]=60
Punkte[1613]=140
Punkte[1614]=70
Punkte[1615]=108
Punkte[1616]=35
Punkte[1617]=127
Punkte[1618]=32
Punkte[1619]=107
Punkte[1620]=31
Punkte[1621]=128
Punkte[1622]=30
Punkte[1623]=133
Punkte[1624]=34
Punkte[1625]=109
Punkte[1626]=173
Punkte[1627]=103
Punkte[1628]=176
Punkte[1629]=77
Punkte[1630]=4
Punkte[1631]=134
Punkte[1632]=179
Punkte[1633]=82
Punkte[1634]=12
Punkte[1635]=80
Punkte[1636]=162
Punkte[1637]=95
Punkte[1638]=21
Punkte[1639]=121
Punkte[1640]=75
Punkte[1641]=172
Punkte[1642]=93
Punkte[1643]=142
Punkte[1644]=64
Punkte[1645]=171
Punkte[1646]=85
Punkte[1647]=178
Punkte[1648]=126
Punkte[1649]=17
Punkte[1650]=151
Punkte[1651]=15
Punkte[1652]=79
Punkte[1653]=6
Punkte[1654]=129
Punkte[1655]=52
Punkte[1656]=167
Punkte[1657]=54
Punkte[1658]=136
Punkte[1659]=83
Punkte[1660]=162
Punkte[1661]=94
Punkte[1662]=143
Punkte[1663]=62
Punkte[1664]=113
Punkte[1665]=18
Punkte[1666]=95
Punkte[1667]=169
Punkte[1668]=63
Punkte[1669]=142
Punkte[1670]=65
Punkte[1671]=164
Punkte[1672]=60
Punkte[1673]=141
Punkte[1674]=72
Punkte[1675]=179
Punkte[1676]=77
Punkte[1677]=171
Punkte[1678]=87
Punkte[1679]=149
Punkte[1680]=117
Punkte[1681]=13
Punkte[1682]=80
Punkte[1683]=23
Punkte[1684]=116
Punkte[1685]=41
Punkte[1686]=106
Punkte[1687]=168
Punkte[1688]=100
Punkte[1689]=166
Punkte[1690]=125
Punkte[1691]=16
Punkte[1692]=86
Punkte[1693]=4
Punkte[1694]=81
Punkte[1695]=9
Punkte[1696]=74
Punkte[1697]=10
Punkte[1698]=78
Punkte[1699]=0
Punkte[1700]=121
Punkte[1701]=72
Punkte[1702]=172
Punkte[1703]=102
Punkte[1704]=19
Punkte[1705]=128
Punkte[1706]=21
Punkte[1707]=93
Punkte[1708]=14
Punkte[1709]=113
Punkte[1710]=12
Punkte[1711]=135
Punkte[1712]=42
Punkte[1713]=104
Punkte[1714]=11
Punkte[1715]=98
Punkte[1716]=170
Punkte[1717]=73
Punkte[1718]=117
Punkte[1719]=173
Punkte[1720]=90
Punkte[1721]=13
Punkte[1722]=95
Punkte[1723]=1
Punkte[1724]=97
Punkte[1725]=7
Punkte[1726]=94
Punkte[1727]=9
Punkte[1728]=116
Punkte[1729]=72
Punkte[1730]=145
Punkte[1731]=77
Punkte[1732]=156
Punkte[1733]=28
Punkte[1734]=134
Punkte[1735]=10
Punkte[1736]=106
Punkte[1737]=140
Punkte[1738]=35
Punkte[1739]=138
Punkte[1740]=87
Punkte[1741]=174
Punkte[1742]=126
Punkte[1743]=21
Punkte[1744]=100
Punkte[1745]=165
Punkte[1746]=78
Punkte[1747]=139
Punkte[1748]=92
Punkte[1749]=168
Punkte[1750]=102
Punkte[1751]=9
Punkte[1752]=86
Punkte[1753]=15
Punkte[1754]=90
Punkte[1755]=5
Punkte[1756]=114
Punkte[1757]=148
Punkte[1758]=77
Punkte[1759]=129
Punkte[1760]=35
Punkte[1761]=130
Punkte[1762]=11
Punkte[1763]=115
Punkte[1764]=39
Punkte[1765]=101
Punkte[1766]=20
Punkte[1767]=132
Punkte[1768]=74
Punkte[1769]=3
Punkte[1770]=75
Punkte[1771]=144
Punkte[1772]=103
Punkte[1773]=38
Punkte[1774]=133
Punkte[1775]=61
Punkte[1776]=142
Punkte[1777]=62
Punkte[1778]=147
Punkte[1779]=14
Punkte[1780]=107
Punkte[1781]=1
Punkte[1782]=80
Punkte[1783]=5
Punkte[1784]=120
Punkte[1785]=177
Punkte[1786]=124
Punkte[1787]=13
Punkte[1788]=82
Punkte[1789]=168
Punkte[1790]=52
Punkte[1791]=132
Punkte[1792]=25
Punkte[1793]=154
Punkte[1794]=24
Punkte[1795]=128
Punkte[1796]=53
Punkte[1797]=136
Punkte[1798]=8
Punkte[1799]=103
Punkte[1800]=37
Punkte[1801]=106
Punkte[1802]=7
Punkte[1803]=58
Punkte[1804]=130
Punkte[1805]=26
Punkte[1806]=171
Punkte[1807]=113
Punkte[1808]=72
Punkte[1809]=10
Punkte[1810]=110
Punkte[1811]=45
Punkte[1812]=146
Punkte[1813]=17
Punkte[1814]=107
Punkte[1815]=3
Punkte[1816]=141
Punkte[1817]=54
Punkte[1818]=142
Punkte[1819]=56
Punkte[1820]=159
Punkte[1821]=92
Punkte[1822]=151
Punkte[1823]=118
Punkte[1824]=150
Punkte[1825]=78
Punkte[1826]=7
Punkte[1827]=136
Punkte[1828]=33
Punkte[1829]=133
Punkte[1830]=177
Punkte[1831]=132
Punkte[1832]=21
Punkte[1833]=124
Punkte[1834]=162
Punkte[1835]=100
Punkte[1836]=4
Punkte[1837]=75
Punkte[1838]=145
Punkte[1839]=87
Punkte[1840]=139
Punkte[1841]=59
Punkte[1842]=135
Punkte[1843]=30
Punkte[1844]=98
Punkte[1845]=20
Punkte[1846]=127
Punkte[1847]=37
Punkte[1848]=141
Punkte[1849]=11
Punkte[1850]=92
Punkte[1851]=12
Punkte[1852]=148
Punkte[1853]=91
Punkte[1854]=8
Punkte[1855]=76
Punkte[1856]=157
Punkte[1857]=18
Punkte[1858]=103
Punkte[1859]=10
Punkte[1860]=95
Punkte[1861]=154
Punkte[1862]=77
Punkte[1863]=130
Punkte[1864]=28
Punkte[1865]=159
Punkte[1866]=69
Punkte[1867]=138
Punkte[1868]=27
Punkte[1869]=104
Punkte[1870]=6
Punkte[1871]=115
Punkte[1872]=70
Punkte[1873]=141
Punkte[1874]=87
Punkte[1875]=5
Punkte[1876]=85
Punkte[1877]=170
Punkte[1878]=57
Punkte[1879]=133
Punkte[1880]=56
Punkte[1881]=124
Punkte[1882]=30
Punkte[1883]=97
Punkte[1884]=165
Punkte[1885]=71
Punkte[1886]=168
Punkte[1887]=83
Punkte[1888]=179
Punkte[1889]=89
Punkte[1890]=23
Punkte[1891]=80
Punkte[1892]=11
Punkte[1893]=82
Punkte[1894]=9
Punkte[1895]=72
Punkte[1896]=117
Punkte[1897]=148
Punkte[1898]=21
Punkte[1899]=98
Punkte[1900]=158
Punkte[1901]=79
Punkte[1902]=14
Punkte[1903]=84
Punkte[1904]=12
Punkte[1905]=100
Punkte[1906]=7
Punkte[1907]=110
Punkte[1908]=35
Punkte[1909]=139
Punkte[1910]=76
Punkte[1911]=162
Punkte[1912]=45
Punkte[1913]=111
Punkte[1914]=175
Punkte[1915]=88
Punkte[1916]=11
Punkte[1917]=77
Punkte[1918]=9
Punkte[1919]=132
Punkte[1920]=24
Punkte[1921]=103
Punkte[1922]=167
Punkte[1923]=50
Punkte[1924]=163
Punkte[1925]=59
Punkte[1926]=142
Punkte[1927]=74
Punkte[1928]=155
Punkte[1929]=22
Punkte[1930]=100
Punkte[1931]=169
Punkte[1932]=89
Punkte[1933]=170
Punkte[1934]=94
Punkte[1935]=14
Punkte[1936]=101
Punkte[1937]=174
Punkte[1938]=78
Punkte[1939]=13
Punkte[1940]=144
Punkte[1941]=66
Punkte[1942]=179
Punkte[1943]=118
Punkte[1944]=28
Punkte[1945]=128
Punkte[1946]=29
Punkte[1947]=156
Punkte[1948]=122
Punkte[1949]=157
Punkte[1950]=83
Punkte[1951]=178
Punkte[1952]=113
Punkte[1953]=177
Punkte[1954]=97
Punkte[1955]=11
Punkte[1956]=99
Punkte[1957]=176
Punkte[1958]=71
Punkte[1959]=173
Punkte[1960]=72
Punkte[1961]=133
Punkte[1962]=77
Punkte[1963]=2
Punkte[1964]=105
Punkte[1965]=51
Punkte[1966]=153
Punkte[1967]=69
Punkte[1968]=137
Punkte[1969]=52
Punkte[1970]=136
Punkte[1971]=24
Punkte[1972]=121
Punkte[1973]=15
Punkte[1974]=79
Punkte[1975]=129
Punkte[1976]=78
Punkte[1977]=161
Punkte[1978]=76
Punkte[1979]=147
Punkte[1980]=112
Punkte[1981]=37
Punkte[1982]=130
Punkte[1983]=56
Punkte[1984]=135
Punkte[1985]=5
Punkte[1986]=89
Punkte[1987]=160
Punkte[1988]=43
Punkte[1989]=105
Punkte[1990]=31
Punkte[1991]=127
Punkte[1992]=175
Punkte[1993]=68
Punkte[1994]=164
Punkte[1995]=62
Punkte[1996]=138
Punkte[1997]=86
Punkte[1998]=161
Punkte[1999]=73
Punkte[2000]=2
Punkte[2001]=84
Punkte[2002]=149
Punkte[2003]=65
Punkte[2004]=141
Punkte[2005]=55
Punkte[2006]=130
Punkte[2007]=59
Punkte[2008]=168
Punkte[2009]=90
Punkte[2010]=143
Punkte[2011]=60
Punkte[2012]=111
Punkte[2013]=46
Punkte[2014]=166
Punkte[2015]=93
Punkte[2016]=18
Punkte[2017]=108
Punkte[2018]=173
Punkte[2019]=124
Punkte[2020]=14
Punkte[2021]=136
Punkte[2022]=79
Punkte[2023]=2
Punkte[2024]=97
Punkte[2025]=26
Punkte[2026]=127
Punkte[2027]=3
Punkte[2028]=133
Punkte[2029]=6
Punkte[2030]=80
Punkte[2031]=139
Punkte[2032]=84
Punkte[2033]=4
Punkte[2034]=101
Punkte[2035]=172
Punkte[2036]=116
Punkte[2037]=40
Punkte[2038]=140
Punkte[2039]=61
Punkte[2040]=137
Punkte[2041]=98
Punkte[2042]=154
Punkte[2043]=19
Punkte[2044]=125
Punkte[2045]=75
Punkte[2046]=120
Punkte[2047]=73
Punkte[2048]=9
Punkte[2049]=70
Punkte[2050]=173
Punkte[2051]=68
Punkte[2052]=152
Punkte[2053]=25
Punkte[2054]=102
Punkte[2055]=175
Punkte[2056]=83
Punkte[2057]=0
Punkte[2058]=134
Punkte[2059]=62
Punkte[2060]=171
Punkte[2061]=114
Punkte[2062]=63
Punkte[2063]=139
Punkte[2064]=67
Punkte[2065]=135
Punkte[2066]=8
Punkte[2067]=107
Punkte[2068]=170
Punkte[2069]=99
Punkte[2070]=167
Punkte[2071]=100
Punkte[2072]=65
Punkte[2073]=132
Punkte[2074]=53
Punkte[2075]=129
Punkte[2076]=30
Punkte[2077]=127
Punkte[2078]=17
Punkte[2079]=156
Punkte[2080]=84
Punkte[2081]=168
Punkte[2082]=77
Punkte[2083]=5
Punkte[2084]=116
Punkte[2085]=67
Punkte[2086]=164
Punkte[2087]=21
Punkte[2088]=131
Punkte[2089]=37
Punkte[2090]=113
Punkte[2091]=15
Punkte[2092]=117
Punkte[2093]=12
Punkte[2094]=111
Punkte[2095]=13
Punkte[2096]=96
Punkte[2097]=18
Punkte[2098]=85
Punkte[2099]=162
Punkte[2100]=48
Punkte[2101]=135
Punkte[2102]=76
Punkte[2103]=10
Punkte[2104]=74
Punkte[2105]=144
Punkte[2106]=79
Punkte[2107]=11
Punkte[2108]=122
Punkte[2109]=22
Punkte[2110]=152
Punkte[2111]=91
Punkte[2112]=14
Punkte[2113]=89
Punkte[2114]=143
Punkte[2115]=86
Punkte[2116]=140
Punkte[2117]=82
Punkte[2118]=33
Punkte[2119]=128
Punkte[2120]=38
Punkte[2121]=102
Punkte[2122]=35
Punkte[2123]=162
Punkte[2124]=49
Punkte[2125]=164
Punkte[2126]=76
Punkte[2127]=119
Punkte[2128]=11
Punkte[2129]=95
Punkte[2130]=9
Punkte[2131]=118
Punkte[2132]=173
Punkte[2133]=75
Punkte[2134]=166
Punkte[2135]=78
Punkte[2136]=179
Punkte[2137]=36
Punkte[2138]=139
Punkte[2139]=92
Punkte[2140]=165
Punkte[2141]=125
Punkte[2142]=26
Punkte[2143]=102
Punkte[2144]=15
Punkte[2145]=96
Punkte[2146]=12
Punkte[2147]=115
Punkte[2148]=148
Punkte[2149]=76
Punkte[2150]=171
Punkte[2151]=88
Punkte[2152]=132
Punkte[2153]=27
Punkte[2154]=129
Punkte[2155]=164
Punkte[2156]=100
Punkte[2157]=173
Punkte[2158]=69
Punkte[2159]=140
Punkte[2160]=2
Punkte[2161]=72
Punkte[2162]=163
Punkte[2163]=77
Punkte[2164]=170
Punkte[2165]=25
Punkte[2166]=128
Punkte[2167]=20
Punkte[2168]=92
Punkte[2169]=166
Punkte[2170]=103
Punkte[2171]=177
Punkte[2172]=81
Punkte[2173]=157
Punkte[2174]=27
Punkte[2175]=123
Punkte[2176]=76
Punkte[2177]=133
Punkte[2178]=83
Punkte[2179]=1
Punkte[2180]=75
Punkte[2181]=171
Punkte[2182]=74
Punkte[2183]=172
Punkte[2184]=80
Punkte[2185]=173
Punkte[2186]=79
Punkte[2187]=160
Punkte[2188]=37
Punkte[2189]=140
Punkte[2190]=64
Punkte[2191]=137
Punkte[2192]=58
Punkte[2193]=144
Punkte[2194]=65
Punkte[2195]=179
Punkte[2196]=71
Punkte[2197]=139
Punkte[2198]=9
Punkte[2199]=78
Punkte[2200]=131
Punkte[2201]=2
Punkte[2202]=98
Punkte[2203]=28
Punkte[2204]=127
Punkte[2205]=18
Punkte[2206]=94
Punkte[2207]=0
Punkte[2208]=107
Punkte[2209]=56
Punkte[2210]=160
Punkte[2211]=57
Punkte[2212]=135
Punkte[2213]=85
Punkte[2214]=149
Punkte[2215]=74
Punkte[2216]=179
Punkte[2217]=75
Punkte[2218]=6
Punkte[2219]=101
Punkte[2220]=38
Punkte[2221]=134
Punkte[2222]=13
Punkte[2223]=141
Punkte[2224]=45
Punkte[2225]=3
Punkte[2226]=90
Punkte[2227]=153
Punkte[2228]=95
Punkte[2229]=161
Punkte[2230]=32
Punkte[2231]=129
Punkte[2232]=76
Punkte[2233]=167
Punkte[2234]=70
Punkte[2235]=176
Punkte[2236]=110
Punkte[2237]=49
Punkte[2238]=150
Punkte[2239]=87
Punkte[2240]=15
Punkte[2241]=112
Punkte[2242]=46
Punkte[2243]=159
Punkte[2244]=85
Punkte[2245]=128
Punkte[2246]=18
Punkte[2247]=126
Punkte[2248]=24
Punkte[2249]=127
Punkte[2250]=19
Punkte[2251]=101
Punkte[2252]=138
Punkte[2253]=66
Punkte[2254]=147
Punkte[2255]=75
Punkte[2256]=134
Punkte[2257]=179
Punkte[2258]=73
Punkte[2259]=0
Punkte[2260]=102
Punkte[2261]=166
Punkte[2262]=47
Punkte[2263]=158
Punkte[2264]=56
Punkte[2265]=132
Punkte[2266]=5
Punkte[2267]=129
Punkte[2268]=8
Punkte[2269]=63
Punkte[2270]=113
Punkte[2271]=11
Punkte[2272]=106
Punkte[2273]=9
Punkte[2274]=110
Punkte[2275]=13
Punkte[2276]=135
Punkte[2277]=82
Punkte[2278]=162
Punkte[2279]=58
Punkte[2280]=139
Punkte[2281]=61
Punkte[2282]=111
Punkte[2283]=147
Punkte[2284]=47
Punkte[2285]=146
Punkte[2286]=36
Punkte[2287]=130
Punkte[2288]=31
Punkte[2289]=142
Punkte[2290]=73
Punkte[2291]=154
Punkte[2292]=86
Punkte[2293]=149
Punkte[2294]=69
Punkte[2295]=123
Punkte[2296]=7
Punkte[2297]=145
Punkte[2298]=10
Punkte[2299]=117
Punkte[2300]=40
Punkte[2301]=104
Punkte[2302]=167
Punkte[2303]=75
Punkte[2304]=8
Punkte[2305]=62
Punkte[2306]=110
Punkte[2307]=168
Punkte[2308]=108
Punkte[2309]=17
Punkte[2310]=114
Punkte[2311]=39
Punkte[2312]=140
Punkte[2313]=67
Punkte[2314]=103
Punkte[2315]=25
Punkte[2316]=152
Punkte[2317]=72
Punkte[2318]=171
Punkte[2319]=77
Punkte[2320]=147
Punkte[2321]=22
Punkte[2322]=96
Punkte[2323]=154
Punkte[2324]=42
Punkte[2325]=155
Punkte[2326]=27
Punkte[2327]=156
Punkte[2328]=30
Punkte[2329]=99
Punkte[2330]=7
Punkte[2331]=114
Punkte[2332]=11
Punkte[2333]=83
Punkte[2334]=10
Punkte[2335]=104
Punkte[2336]=68
Punkte[2337]=120
Punkte[2338]=76
Punkte[2339]=173
Punkte[2340]=81
Punkte[2341]=143
Punkte[2342]=14
Punkte[2343]=79
Punkte[2344]=16
Punkte[2345]=88
Punkte[2346]=147
Punkte[2347]=72
Punkte[2348]=124
Punkte[2349]=12
Punkte[2350]=122
Punkte[2351]=157
Punkte[2352]=77
Punkte[2353]=8
Punkte[2354]=134
Punkte[2355]=49
Punkte[2356]=152
Punkte[2357]=50
Punkte[2358]=151
Punkte[2359]=64
Punkte[2360]=136
Punkte[2361]=29
Punkte[2362]=131
Punkte[2363]=63
Punkte[2364]=137
Punkte[2365]=30
Punkte[2366]=100
Punkte[2367]=163
Punkte[2368]=92
Punkte[2369]=167
Punkte[2370]=98
Punkte[2371]=17
Punkte[2372]=113
Punkte[2373]=47
Punkte[2374]=4
Punkte[2375]=78
Punkte[2376]=175
Punkte[2377]=105
Punkte[2378]=39
Punkte[2379]=107
Punkte[2380]=12
Punkte[2381]=104
Punkte[2382]=8
Punkte[2383]=76
Punkte[2384]=11
Punkte[2385]=87
Punkte[2386]=6
Punkte[2387]=88
Punkte[2388]=7
Punkte[2389]=125
Punkte[2390]=72
Punkte[2391]=143
Punkte[2392]=68
Punkte[2393]=169
Punkte[2394]=80
Punkte[2395]=133
Punkte[2396]=34
Punkte[2397]=100
Punkte[2398]=3
Punkte[2399]=73
Punkte[2400]=174
Punkte[2401]=105
Punkte[2402]=41
Punkte[2403]=117
Punkte[2404]=148
Punkte[2405]=12
Punkte[2406]=83
Punkte[2407]=4
Punkte[2408]=90
Punkte[2409]=170
Punkte[2410]=93
Punkte[2411]=176
Punkte[2412]=102
Punkte[2413]=5
Punkte[2414]=109
Punkte[2415]=33
Punkte[2416]=131
Punkte[2417]=36
Punkte[2418]=154
Punkte[2419]=78
Punkte[2420]=128
Punkte[2421]=43
Punkte[2422]=165
Punkte[2423]=81
Punkte[2424]=28
Punkte[2425]=126
Punkte[2426]=2
Punkte[2427]=91
Punkte[2428]=56
Punkte[2429]=167
Punkte[2430]=49
Punkte[2431]=151
Punkte[2432]=77
Punkte[2433]=153
Punkte[2434]=121
Punkte[2435]=177
Punkte[2436]=133
Punkte[2437]=10
Punkte[2438]=100
Punkte[2439]=35
Punkte[2440]=135
Punkte[2441]=14
Punkte[2442]=111
Punkte[2443]=170
Punkte[2444]=82
Punkte[2445]=178
Punkte[2446]=125
Punkte[2447]=22
Punkte[2448]=166
Punkte[2449]=130
Punkte[2450]=24
Punkte[2451]=138
Punkte[2452]=5
Punkte[2453]=76
Punkte[2454]=124
Punkte[2455]=7
Punkte[2456]=145
Punkte[2457]=61
Punkte[2458]=95
Punkte[2459]=16
Punkte[2460]=99
Punkte[2461]=26
Punkte[2462]=132
Punkte[2463]=52
Punkte[2464]=121
Punkte[2465]=43
Punkte[2466]=122
Punkte[2467]=25
Punkte[2468]=125
Punkte[2469]=23
Punkte[2470]=98
Punkte[2471]=174
Punkte[2472]=74
Punkte[2473]=3
Punkte[2474]=44
Punkte[2475]=141
Punkte[2476]=89
Punkte[2477]=164
Punkte[2478]=75
Punkte[2479]=152
Punkte[2480]=69
Punkte[2481]=176
Punkte[2482]=84
Punkte[2483]=14
Punkte[2484]=107
Punkte[2485]=11
Punkte[2486]=140
Punkte[2487]=72
Punkte[2488]=142
Punkte[2489]=58
Punkte[2490]=112
Punkte[2491]=9
Punkte[2492]=103
Punkte[2493]=169
Punkte[2494]=99
Punkte[2495]=165
Punkte[2496]=51
Punkte[2497]=108
Punkte[2498]=33
Punkte[2499]=159
Punkte[2500]=86
Punkte[2501]=129
Punkte[2502]=18
Punkte[2503]=95
Punkte[2504]=0
Punkte[2505]=137
Punkte[2506]=62
Punkte[2507]=139
Punkte[2508]=64
Punkte[2509]=173
Punkte[2510]=96
Punkte[2511]=163
Punkte[2512]=97
Punkte[2513]=168
Punkte[2514]=55
Punkte[2515]=160
Punkte[2516]=70
Punkte[2517]=109
Punkte[2518]=21
Punkte[2519]=115
Punkte[2520]=11
Punkte[2521]=108
Punkte[2522]=10
Punkte[2523]=73
Punkte[2524]=143
Punkte[2525]=66
Punkte[2526]=179
Punkte[2527]=128
Punkte[2528]=2
Punkte[2529]=125
Punkte[2530]=24
Punkte[2531]=151
Punkte[2532]=67
Punkte[2533]=120
Punkte[2534]=4
Punkte[2535]=77
Punkte[2536]=131
Punkte[2537]=39
Punkte[2538]=135
Punkte[2539]=7
Punkte[2540]=110
Punkte[2541]=56
Punkte[2542]=168
Punkte[2543]=54
Punkte[2544]=166
Punkte[2545]=97
Punkte[2546]=12
Punkte[2547]=105
Punkte[2548]=29
Punkte[2549]=99
Punkte[2550]=30
Punkte[2551]=175
Punkte[2552]=69
Punkte[2553]=141
Punkte[2554]=55
Punkte[2555]=109
Punkte[2556]=44
Punkte[2557]=145
Punkte[2558]=81
Punkte[2559]=27
Punkte[2560]=128
Punkte[2561]=1
Punkte[2562]=73
Punkte[2563]=123
Punkte[2564]=46
Punkte[2565]=156
Punkte[2566]=91
Punkte[2567]=25
Punkte[2568]=101
Punkte[2569]=36
Punkte[2570]=129
Punkte[2571]=0
Punkte[2572]=77
Punkte[2573]=143
Punkte[2574]=40
Punkte[2575]=134
Punkte[2576]=15
Punkte[2577]=89
Punkte[2578]=22
Punkte[2579]=136
Punkte[2580]=68
Punkte[2581]=144
Punkte[2582]=71
Punkte[2583]=151
Punkte[2584]=41
Punkte[2585]=164
Punkte[2586]=74
Punkte[2587]=9
Punkte[2588]=130
Punkte[2589]=32
Punkte[2590]=127
Punkte[2591]=29
Punkte[2592]=156
Punkte[2593]=44
Punkte[2594]=106
Punkte[2595]=30
Punkte[2596]=132
Punkte[2597]=172
Punkte[2598]=96
Punkte[2599]=3
Punkte[2600]=89
Punkte[2601]=163
Punkte[2602]=82
Punkte[2603]=13
Punkte[2604]=80
Punkte[2605]=165
Punkte[2606]=95
Punkte[2607]=178
Punkte[2608]=79
Punkte[2609]=133
Punkte[2610]=57
Punkte[2611]=138
Punkte[2612]=64
Punkte[2613]=115
Punkte[2614]=5
Punkte[2615]=51
Punkte[2616]=135
Punkte[2617]=41
Punkte[2618]=149
Punkte[2619]=116
Punkte[2620]=6
Punkte[2621]=117
Punkte[2622]=8
Punkte[2623]=100
Punkte[2624]=171
Punkte[2625]=86
Punkte[2626]=167
Punkte[2627]=83
Punkte[2628]=151
Punkte[2629]=22
Punkte[2630]=133
Punkte[2631]=82
Punkte[2632]=164
Punkte[2633]=95
Punkte[2634]=14
Punkte[2635]=119
Punkte[2636]=174
Punkte[2637]=65
Punkte[2638]=163
Punkte[2639]=66
Punkte[2640]=170
Punkte[2641]=74
Punkte[2642]=10
Punkte[2643]=76
Punkte[2644]=130
Punkte[2645]=23
Punkte[2646]=122
Punkte[2647]=75
Punkte[2648]=2
Punkte[2649]=101
Punkte[2650]=9
Punkte[2651]=70
Punkte[2652]=132
Punkte[2653]=38
Punkte[2654]=140
Punkte[2655]=87
Punkte[2656]=48
Punkte[2657]=160
Punkte[2658]=88
Punkte[2659]=19
Punkte[2660]=105
Punkte[2661]=11
Punkte[2662]=98
Punkte[2663]=164
Punkte[2664]=64
Punkte[2665]=137
Punkte[2666]=79
Punkte[2667]=177
Punkte[2668]=74
Punkte[2669]=173
Punkte[2670]=72
Punkte[2671]=9
Punkte[2672]=133
Punkte[2673]=81
Punkte[2674]=134
Punkte[2675]=59
Punkte[2676]=142
Punkte[2677]=94
Punkte[2678]=143
Punkte[2679]=61
Punkte[2680]=135
Punkte[2681]=33
Punkte[2682]=105
Punkte[2683]=3
Punkte[2684]=83
Punkte[2685]=154
Punkte[2686]=121
Punkte[2687]=50
Punkte[2688]=120
Punkte[2689]=153
Punkte[2690]=18
Punkte[2691]=85
Punkte[2692]=169
Punkte[2693]=86
Punkte[2694]=166
Punkte[2695]=69
Punkte[2696]=145
Punkte[2697]=16
Punkte[2698]=80
Punkte[2699]=168
Punkte[2700]=79
Punkte[2701]=162
Punkte[2702]=95
Punkte[2703]=19
Punkte[2704]=93
Punkte[2705]=21
Punkte[2706]=155
Punkte[2707]=45
Punkte[2708]=103
Punkte[2709]=46
Punkte[2710]=129
Punkte[2711]=35
Punkte[2712]=146
Punkte[2713]=63
Punkte[2714]=144
Punkte[2715]=70
Punkte[2716]=172
Punkte[2717]=122
Punkte[2718]=22
Punkte[2719]=156
Punkte[2720]=17
Punkte[2721]=107
Punkte[2722]=179
Punkte[2723]=117
Punkte[2724]=10
Punkte[2725]=72
Punkte[2726]=4
Punkte[2727]=118
Punkte[2728]=13
Punkte[2729]=78
Punkte[2730]=131
Punkte[2731]=19
Punkte[2732]=130
Punkte[2733]=26
Punkte[2734]=103
Punkte[2735]=38
Punkte[2736]=148
Punkte[2737]=68
Punkte[2738]=105
Punkte[2739]=40
Punkte[2740]=84
Punkte[2741]=5
Punkte[2742]=79
Punkte[2743]=150
Punkte[2744]=91
Punkte[2745]=141
Punkte[2746]=90
Punkte[2747]=12
Punkte[2748]=128
Punkte[2749]=10
Punkte[2750]=78
Punkte[2751]=161
Punkte[2752]=66
Punkte[2753]=157
Punkte[2754]=18
Punkte[2755]=80
Punkte[2756]=158
Punkte[2757]=85
Punkte[2758]=15
Punkte[2759]=114
Punkte[2760]=19
Punkte[2761]=103
Punkte[2762]=39
Punkte[2763]=148
Punkte[2764]=48
Punkte[2765]=116
Punkte[2766]=170
Punkte[2767]=86
Punkte[2768]=165
Punkte[2769]=89
Punkte[2770]=134
Punkte[2771]=83
Punkte[2772]=133
Punkte[2773]=37
Punkte[2774]=163
Punkte[2775]=60
Punkte[2776]=142
Punkte[2777]=57
Punkte[2778]=169
Punkte[2779]=78
Punkte[2780]=152
Punkte[2781]=24
Punkte[2782]=131
Punkte[2783]=61
Punkte[2784]=154
Punkte[2785]=123
Punkte[2786]=55
Punkte[2787]=167
Punkte[2788]=77
Punkte[2789]=149
Punkte[2790]=91
Punkte[2791]=17
Punkte[2792]=102
Punkte[2793]=36
Punkte[2794]=157
Punkte[2795]=79
Punkte[2796]=158
Punkte[2797]=75
Punkte[2798]=174
Punkte[2799]=100
Punkte[2800]=168
Punkte[2801]=85
Punkte[2802]=176
Punkte[2803]=31
Punkte[2804]=129
Punkte[2805]=32
Punkte[2806]=133
Punkte[2807]=61
Punkte[2808]=142
Punkte[2809]=83
Punkte[2810]=15
Punkte[2811]=94
Punkte[2812]=28
Punkte[2813]=106
Punkte[2814]=10
Punkte[2815]=118
Punkte[2816]=22
Punkte[2817]=138
Punkte[2818]=73
Punkte[2819]=170
Punkte[2820]=69
Punkte[2821]=9
Punkte[2822]=98
Punkte[2823]=154
Punkte[2824]=77
Punkte[2825]=165
Punkte[2826]=97
Punkte[2827]=3
Punkte[2828]=82
Punkte[2829]=0
Punkte[2830]=71
Punkte[2831]=175
Punkte[2832]=53
Punkte[2833]=128
Punkte[2834]=34
Punkte[2835]=153
Punkte[2836]=41
Punkte[2837]=110
Punkte[2838]=37
Punkte[2839]=100
Punkte[2840]=166
Punkte[2841]=65
Punkte[2842]=172
Punkte[2843]=87
Punkte[2844]=20
Punkte[2845]=127
Punkte[2846]=81
Punkte[2847]=7
Punkte[2848]=145
Punkte[2849]=59
Punkte[2850]=113
Punkte[2851]=177
Punkte[2852]=67
Punkte[2853]=0
Punkte[2854]=106
Punkte[2855]=140
Punkte[2856]=62
Punkte[2857]=150
Punkte[2858]=15
Punkte[2859]=92
Punkte[2860]=138
Punkte[2861]=68
Punkte[2862]=146
Punkte[2863]=95
Punkte[2864]=26
Punkte[2865]=129
Punkte[2866]=52
Punkte[2867]=127
Punkte[2868]=160
Punkte[2869]=77
Punkte[2870]=152
Punkte[2871]=91
Punkte[2872]=3
Punkte[2873]=75
Punkte[2874]=134
Punkte[2875]=7
Punkte[2876]=114
Punkte[2877]=0
Punkte[2878]=100
Punkte[2879]=18
Punkte[2880]=135
Punkte[2881]=55
Punkte[2882]=6
Punkte[2883]=119
Punkte[2884]=16
Punkte[2885]=137
Punkte[2886]=23
Punkte[2887]=131
Punkte[2888]=64
Punkte[2889]=140
Punkte[2890]=15
Punkte[2891]=143
Punkte[2892]=58
Punkte[2893]=177
Punkte[2894]=87
Punkte[2895]=12
Punkte[2896]=78
Punkte[2897]=155
Punkte[2898]=93
Punkte[2899]=179
Punkte[2900]=72
Punkte[2901]=147
Punkte[2902]=14
Punkte[2903]=144
Punkte[2904]=44
Punkte[2905]=161
Punkte[2906]=73
Punkte[2907]=173
Punkte[2908]=77
Punkte[2909]=129
Punkte[2910]=34
Punkte[2911]=98
Punkte[2912]=29
Punkte[2913]=158
Punkte[2914]=91
Punkte[2915]=151
Punkte[2916]=94
Punkte[2917]=17
Punkte[2918]=83
Punkte[2919]=157
Punkte[2920]=30
Punkte[2921]=156
Punkte[2922]=125
Punkte[2923]=72
Punkte[2924]=2
Punkte[2925]=140
Punkte[2926]=107
Punkte[2927]=56
Punkte[2928]=176
Punkte[2929]=63
Punkte[2930]=136
Punkte[2931]=58
Punkte[2932]=139
Punkte[2933]=59
Punkte[2934]=144
Punkte[2935]=87
Punkte[2936]=168
Punkte[2937]=88
Punkte[2938]=14
Punkte[2939]=79
Punkte[2940]=141
Punkte[2941]=60
Punkte[2942]=171
Punkte[2943]=68
Punkte[2944]=131
Punkte[2945]=9
Punkte[2946]=110
Punkte[2947]=53
Punkte[2948]=122
Punkte[2949]=11
Punkte[2950]=76
Punkte[2951]=119
Punkte[2952]=0
Punkte[2953]=37
Punkte[2954]=83
Punkte[2955]=2
Punkte[2956]=133
Punkte[2957]=10
Punkte[2958]=43
Punkte[2959]=145
Punkte[2960]=86
Punkte[2961]=4
Punkte[2962]=87
Punkte[2963]=159
Punkte[2964]=80
Punkte[2965]=7
Punkte[2966]=95
Punkte[2967]=20
Punkte[2968]=103
Punkte[2969]=172
Punkte[2970]=104
Punkte[2971]=21
Punkte[2972]=147
Punkte[2973]=68
Punkte[2974]=125
Punkte[2975]=31
Punkte[2976]=96
Punkte[2977]=5
Punkte[2978]=108
Punkte[2979]=8
Punkte[2980]=84
Punkte[2981]=14
Punkte[2982]=85
Punkte[2983]=178
Punkte[2984]=112
Punkte[2985]=26
Punkte[2986]=90
Punkte[2987]=179
Punkte[2988]=71
Punkte[2989]=146
Punkte[2990]=78
Punkte[2991]=166
Punkte[2992]=64
Punkte[2993]=165
Punkte[2994]=65
Punkte[2995]=149
Punkte[2996]=76
Punkte[2997]=155
Punkte[2998]=43
Punkte[2999]=10
Punkte[3000]=102
Punkte[3001]=168
Punkte[3002]=105
Punkte[3003]=18
Punkte[3004]=80
Punkte[3005]=21
Punkte[3006]=154
Punkte[3007]=16
Punkte[3008]=124
Punkte[3009]=28
Punkte[3010]=133
Punkte[3011]=60
Punkte[3012]=143
Punkte[3013]=71
Punkte[3014]=119
Punkte[3015]=22
Punkte[3016]=104
Punkte[3017]=9
Punkte[3018]=103
Punkte[3019]=27
Punkte[3020]=139
Punkte[3021]=41
Punkte[3022]=150
Punkte[3023]=74
Punkte[3024]=169
Punkte[3025]=67
Punkte[3026]=151
Punkte[3027]=65
Punkte[3028]=141
Punkte[3029]=12
Punkte[3030]=124
Punkte[3031]=20
Punkte[3032]=148
Punkte[3033]=44
Punkte[3034]=97
Punkte[3035]=164
Punkte[3036]=94
Punkte[3037]=5
Punkte[3038]=85
Punkte[3039]=175
Punkte[3040]=111
Punkte[3041]=42
Punkte[3042]=153
Punkte[3043]=16
Punkte[3044]=79
Punkte[3045]=139
Punkte[3046]=78
Punkte[3047]=14
Punkte[3048]=127
Punkte[3049]=27
Punkte[3050]=117
Punkte[3051]=68
Punkte[3052]=172
Punkte[3053]=66
Punkte[3054]=174
Punkte[3055]=118
Punkte[3056]=18
Punkte[3057]=129
Punkte[3058]=51
Punkte[3059]=131
Punkte[3060]=55
Punkte[3061]=140
Punkte[3062]=42
Punkte[3063]=128
Punkte[3064]=178
Punkte[3065]=101
Punkte[3066]=8
Punkte[3067]=97
Punkte[3068]=167
Punkte[3069]=88
Punkte[3070]=17
Punkte[3071]=80
Punkte[3072]=164
Punkte[3073]=99
Punkte[3074]=162
Punkte[3075]=48
Punkte[3076]=158
Punkte[3077]=65
Punkte[3078]=142
Punkte[3079]=16
Punkte[3080]=83
Punkte[3081]=6
Punkte[3082]=115
Punkte[3083]=3
Punkte[3084]=74
Punkte[3085]=10
Punkte[3086]=140
Punkte[3087]=76
Punkte[3088]=153
Punkte[3089]=95
Punkte[3090]=172
Punkte[3091]=102
Punkte[3092]=67
Punkte[3093]=170
Punkte[3094]=25
Punkte[3095]=100
Punkte[3096]=164
Punkte[3097]=92
Punkte[3098]=1
Punkte[3099]=69
Punkte[3100]=141
Punkte[3101]=17
Punkte[3102]=122
Punkte[3103]=45
Punkte[3104]=162
Punkte[3105]=57
Punkte[3106]=142
Punkte[3107]=86
Punkte[3108]=7
Punkte[3109]=58
Punkte[3110]=80
Punkte[3111]=138
Punkte[3112]=101
Punkte[3113]=6
Punkte[3114]=131
Punkte[3115]=36
Punkte[3116]=134
Punkte[3117]=26
Punkte[3118]=124
Punkte[3119]=30
Punkte[3120]=128
Punkte[3121]=12
Punkte[3122]=102
Punkte[3123]=35
Punkte[3124]=133
Punkte[3125]=62
Punkte[3126]=112
Punkte[3127]=59
Punkte[3128]=162
Punkte[3129]=76
Punkte[3130]=161
Punkte[3131]=65
Punkte[3132]=100
Punkte[3133]=138
Punkte[3134]=87
Punkte[3135]=175
Punkte[3136]=90
Punkte[3137]=144
Punkte[3138]=77
Punkte[3139]=130
Punkte[3140]=26
Punkte[3141]=158
Punkte[3142]=56
Punkte[3143]=134
Punkte[3144]=28
Punkte[3145]=155
Punkte[3146]=61
Punkte[3147]=131
Punkte[3148]=54
Punkte[3149]=128
Punkte[3150]=64
Punkte[3151]=171
Punkte[3152]=60
Punkte[3153]=145
Punkte[3154]=46
Punkte[3155]=137
Punkte[3156]=27
Punkte[3157]=95
Punkte[3158]=179
Punkte[3159]=127
Punkte[3160]=30
Punkte[3161]=159
Punkte[3162]=79
Punkte[3163]=147
Punkte[3164]=47
Punkte[3165]=161
Punkte[3166]=71
Punkte[3167]=0
Punkte[3168]=108
Punkte[3169]=11
Punkte[3170]=146
Punkte[3171]=24
Punkte[3172]=128
Punkte[3173]=31
Punkte[3174]=130
Punkte[3175]=87
Punkte[3176]=13
Punkte[3177]=121
Punkte[3178]=52
Punkte[3179]=135
Punkte[3180]=6
Punkte[3181]=84
Punkte[3182]=15
Punkte[3183]=93
Punkte[3184]=18
Punkte[3185]=96
Punkte[3186]=43
Punkte[3187]=10
Punkte[3188]=74
Punkte[3189]=120
Punkte[3190]=76
Punkte[3191]=143
Punkte[3192]=73
Punkte[3193]=9
Punkte[3194]=70
Punkte[3195]=163
Punkte[3196]=38
Punkte[3197]=149
Punkte[3198]=21
Punkte[3199]=164
Punkte[3200]=48
Punkte[3201]=160
Punkte[3202]=94
Punkte[3203]=19
Punkte[3204]=116
Punkte[3205]=5
Punkte[3206]=138
Punkte[3207]=85
Punkte[3208]=142
Punkte[3209]=4
Punkte[3210]=74
Punkte[3211]=141
Punkte[3212]=83
Punkte[3213]=179
Punkte[3214]=123
Punkte[3215]=159
Punkte[3216]=78
Punkte[3217]=131
Punkte[3218]=50
Punkte[3219]=166
Punkte[3220]=75
Punkte[3221]=169
Punkte[3222]=68
Punkte[3223]=162
Punkte[3224]=88
Punkte[3225]=13
Punkte[3226]=97
Punkte[3227]=12
Punkte[3228]=106
Punkte[3229]=145
Punkte[3230]=87
Punkte[3231]=19
Punkte[3232]=96
Punkte[3233]=155
Punkte[3234]=26
Punkte[3235]=153
Punkte[3236]=24
Punkte[3237]=109
Punkte[3238]=22
Punkte[3239]=101
Punkte[3240]=36
Punkte[3241]=105
Punkte[3242]=45
Punkte[3243]=163
Punkte[3244]=60
Punkte[3245]=144
Punkte[3246]=74
Punkte[3247]=121
Punkte[3248]=5
Punkte[3249]=73
Punkte[3250]=172
Punkte[3251]=71
Punkte[3252]=174
Punkte[3253]=99
Punkte[3254]=170
Punkte[3255]=100
Punkte[3256]=30
Punkte[3257]=97
Punkte[3258]=10
Punkte[3259]=127
Punkte[3260]=38
Punkte[3261]=137
Punkte[3262]=76
Punkte[3263]=1
Punkte[3264]=96
Punkte[3265]=2
Punkte[3266]=93
Punkte[3267]=152
Punkte[3268]=81
Punkte[3269]=27
Punkte[3270]=122
Punkte[3271]=12
Punkte[3272]=104
Punkte[3273]=43
Punkte[3274]=144
Punkte[3275]=72
Punkte[3276]=160
Punkte[3277]=46
Punkte[3278]=111
Punkte[3279]=59
Punkte[3280]=133
Punkte[3281]=7
Punkte[3282]=121
Punkte[3283]=11
Punkte[3284]=135
Punkte[3285]=23
Punkte[3286]=149
Punkte[3287]=64
Punkte[3288]=176
Punkte[3289]=56
Punkte[3290]=129
Punkte[3291]=37
Punkte[3292]=132
Punkte[3293]=77
Punkte[3294]=145
Punkte[3295]=95
Punkte[3296]=161
Punkte[3297]=85
Punkte[3298]=136
Punkte[3299]=42
Punkte[3300]=138
Punkte[3301]=86
Punkte[3302]=174
Punkte[3303]=69
Punkte[3304]=147
Punkte[3305]=12
Punkte[3306]=121
Punkte[3307]=6
Punkte[3308]=106
Punkte[3309]=168
Punkte[3310]=78
Punkte[3311]=157
Punkte[3312]=125
Punkte[3313]=164
Punkte[3314]=91
Punkte[3315]=150
Punkte[3316]=14
Punkte[3317]=102
Punkte[3318]=5
Punkte[3319]=115
Punkte[3320]=40
Punkte[3321]=113
Punkte[3322]=148
Punkte[3323]=81
Punkte[3324]=163
Punkte[3325]=64
Punkte[3326]=111
Punkte[3327]=31
Punkte[3328]=176
Punkte[3329]=106
Punkte[3330]=4
Punkte[3331]=105
Punkte[3332]=39
Punkte[3333]=101
Punkte[3334]=35
Punkte[3335]=107
Punkte[3336]=26
Punkte[3337]=133
Punkte[3338]=75
Punkte[3339]=178
Punkte[3340]=118
Punkte[3341]=9
Punkte[3342]=119
Punkte[3343]=10
Punkte[3344]=73
Punkte[3345]=2
Punkte[3346]=100
Punkte[3347]=16
Punkte[3348]=79
Punkte[3349]=48
Punkte[3350]=123
Punkte[3351]=74
Punkte[3352]=179
Punkte[3353]=128
Punkte[3354]=6
Punkte[3355]=132
Punkte[3356]=24
Punkte[3357]=139
Punkte[3358]=64
Punkte[3359]=165
Punkte[3360]=91
Punkte[3361]=57
Punkte[3362]=144
Punkte[3363]=84
Punkte[3364]=158
Punkte[3365]=81
Punkte[3366]=176
Punkte[3367]=129
Punkte[3368]=49
Punkte[3369]=166
Punkte[3370]=67
Punkte[3371]=162
Punkte[3372]=98
Punkte[3373]=153
Punkte[3374]=63
Punkte[3375]=8
Punkte[3376]=75
Punkte[3377]=173
Punkte[3378]=107
Punkte[3379]=23
Punkte[3380]=115
Punkte[3381]=16
Punkte[3382]=89
Punkte[3383]=22
Punkte[3384]=120
Punkte[3385]=69
Punkte[3386]=175
Punkte[3387]=70
Punkte[3388]=172
Punkte[3389]=132
Punkte[3390]=74
Punkte[3391]=9
Punkte[3392]=72
Punkte[3393]=152
Punkte[3394]=25
Punkte[3395]=127
Punkte[3396]=12
Punkte[3397]=137
Punkte[3398]=56
Punkte[3399]=116
Punkte[3400]=34
Punkte[3401]=131
Punkte[3402]=176
Punkte[3403]=104
Punkte[3404]=40
Punkte[3405]=140
Punkte[3406]=29
Punkte[3407]=124
Punkte[3408]=28
Punkte[3409]=130
Punkte[3410]=78
Punkte[3411]=132
Punkte[3412]=66
Punkte[3413]=145
Punkte[3414]=90
Punkte[3415]=7
Punkte[3416]=88
Punkte[3417]=177
Punkte[3418]=92
Punkte[3419]=15
Punkte[3420]=79
Punkte[3421]=158
Punkte[3422]=32
Punkte[3423]=109
Punkte[3424]=179
Punkte[3425]=91
Punkte[3426]=16
Punkte[3427]=99
Punkte[3428]=9
Punkte[3429]=136
Punkte[3430]=23
Punkte[3431]=96
Punkte[3432]=5
Punkte[3433]=135
Punkte[3434]=62
Punkte[3435]=145
Punkte[3436]=45
Punkte[3437]=154
Punkte[3438]=72
Punkte[3439]=147
Punkte[3440]=64
Punkte[3441]=177
Punkte[3442]=113
Punkte[3443]=15
Punkte[3444]=141
Punkte[3445]=55
Punkte[3446]=166
Punkte[3447]=69
Punkte[3448]=0
Punkte[3449]=77
Punkte[3450]=143
Punkte[3451]=19
Punkte[3452]=79
Punkte[3453]=165
Punkte[3454]=44
Punkte[3455]=97
Punkte[3456]=163
Punkte[3457]=76
Punkte[3458]=3
Punkte[3459]=74
Punkte[3460]=127
Punkte[3461]=32
Punkte[3462]=98
Punkte[3463]=156
Punkte[3464]=90
Punkte[3465]=170
Punkte[3466]=83
Punkte[3467]=9
Punkte[3468]=130
Punkte[3469]=56
Punkte[3470]=138
Punkte[3471]=65
Punkte[3472]=161
Punkte[3473]=96
Punkte[3474]=43
Punkte[3475]=10
Punkte[3476]=136
Punkte[3477]=35
Punkte[3478]=108
Punkte[3479]=39
Punkte[3480]=131
Punkte[3481]=60
Punkte[3482]=163
Punkte[3483]=82
Punkte[3484]=179
Punkte[3485]=94
Punkte[3486]=14
Punkte[3487]=113
Punkte[3488]=59
Punkte[3489]=142
Punkte[3490]=75
Punkte[3491]=151
Punkte[3492]=92
Punkte[3493]=162
Punkte[3494]=99
Punkte[3495]=30
Punkte[3496]=130
Punkte[3497]=51
Punkte[3498]=167
Punkte[3499]=70
Punkte[3500]=3
Punkte[3501]=77
Punkte[3502]=156
Punkte[3503]=34
Punkte[3504]=122
Punkte[3505]=54
Punkte[3506]=138
Punkte[3507]=84
Punkte[3508]=14
Punkte[3509]=86
Punkte[3510]=11
Punkte[3511]=101
Punkte[3512]=20
Punkte[3513]=143
Punkte[3514]=57
Punkte[3515]=118
Punkte[3516]=21
Punkte[3517]=155
Punkte[3518]=45
Punkte[3519]=141
Punkte[3520]=17
Punkte[3521]=136
Punkte[3522]=179
Punkte[3523]=72
Punkte[3524]=10
Punkte[3525]=106
Punkte[3526]=178
Punkte[3527]=125
Punkte[3528]=8
Punkte[3529]=137
Punkte[3530]=40
Punkte[3531]=93
Punkte[3532]=162
Punkte[3533]=71
Punkte[3534]=171
Punkte[3535]=100
Punkte[3536]=175
Punkte[3537]=74
Punkte[3538]=119
Punkte[3539]=0
Punkte[3540]=66
Punkte[3541]=157
Punkte[3542]=31
Punkte[3543]=111
Punkte[3544]=169
Punkte[3545]=103
Punkte[3546]=20
Punkte[3547]=123
Punkte[3548]=14
Punkte[3549]=105
Punkte[3550]=11
Punkte[3551]=142
Punkte[3552]=83
Punkte[3553]=134
Punkte[3554]=30
Punkte[3555]=128
Punkte[3556]=10
Punkte[3557]=130
Punkte[3558]=13
Punkte[3559]=98
Punkte[3560]=19
Punkte[3561]=106
Punkte[3562]=22
Punkte[3563]=136
Punkte[3564]=60
Punkte[3565]=139
Punkte[3566]=68
Punkte[3567]=154
Punkte[3568]=34
Punkte[3569]=137
Punkte[3570]=42
Punkte[3571]=135
Punkte[3572]=81
Punkte[3573]=140
Punkte[3574]=87
Punkte[3575]=6
Punkte[3576]=76
Punkte[3577]=127
Punkte[3578]=33
Punkte[3579]=102
Punkte[3580]=36
Punkte[3581]=130
Punkte[3582]=24
Punkte[3583]=108
Punkte[3584]=55
Punkte[3585]=159
Punkte[3586]=38
Punkte[3587]=101
Punkte[3588]=178
Punkte[3589]=72
Punkte[3590]=1
Punkte[3591]=68
Punkte[3592]=124
Punkte[3593]=47
Punkte[3594]=165
Punkte[3595]=86
Punkte[3596]=13
Punkte[3597]=143
Punkte[3598]=81
Punkte[3599]=171
Punkte[3600]=44
Punkte[3601]=131
Punkte[3602]=76
Punkte[3603]=11
Punkte[3604]=100
Punkte[3605]=168
Punkte[3606]=92
Punkte[3607]=139
Punkte[3608]=73
Punkte[3609]=161
Punkte[3610]=74
Punkte[3611]=152
Punkte[3612]=26
Punkte[3613]=129
Punkte[3614]=21
Punkte[3615]=80
Punkte[3616]=58
Punkte[3617]=135
Punkte[3618]=48
Punkte[3619]=163
Punkte[3620]=94
Punkte[3621]=25
Punkte[3622]=109
Punkte[3623]=36
Punkte[3624]=154
Punkte[3625]=16
Punkte[3626]=97
Punkte[3627]=162
Punkte[3628]=63
Punkte[3629]=147
Punkte[3630]=95
Punkte[3631]=174
Punkte[3632]=117
Punkte[3633]=8
Punkte[3634]=89
Punkte[3635]=160
Punkte[3636]=64
Punkte[3637]=172
Punkte[3638]=72
Punkte[3639]=115
Punkte[3640]=48
Punkte[3641]=79
Punkte[3642]=135
Punkte[3643]=45
Punkte[3644]=126
Punkte[3645]=49
Punkte[3646]=136
Punkte[3647]=4
Punkte[3648]=142
Punkte[3649]=58
Punkte[3650]=141
Punkte[3651]=108
Punkte[3652]=0
Punkte[3653]=91
Punkte[3654]=149
Punkte[3655]=78
Punkte[3656]=123
Punkte[3657]=176
Punkte[3658]=100
Punkte[3659]=164
Punkte[3660]=76
Punkte[3661]=10
Punkte[3662]=44
Punkte[3663]=146
Punkte[3664]=75
Punkte[3665]=118
Punkte[3666]=62
Punkte[3667]=154
Punkte[3668]=71
Punkte[3669]=173
Punkte[3670]=104
Punkte[3671]=46
Punkte[3672]=124
Punkte[3673]=26
Punkte[3674]=130
Punkte[3675]=23
Punkte[3676]=125
Punkte[3677]=55
Punkte[3678]=152
Punkte[3679]=68
Punkte[3680]=106
Punkte[3681]=11
Punkte[3682]=94
Punkte[3683]=8
Punkte[3684]=69
Punkte[3685]=107
Punkte[3686]=31
Punkte[3687]=133
Punkte[3688]=50
Punkte[3689]=153
Punkte[3690]=40
Punkte[3691]=139
Punkte[3692]=64
Punkte[3693]=5
Punkte[3694]=96
Punkte[3695]=17
Punkte[3696]=156
Punkte[3697]=44
Punkte[3698]=115
Punkte[3699]=174
Punkte[3700]=87
Punkte[3701]=158
Punkte[3702]=29
Punkte[3703]=151
Punkte[3704]=79
Punkte[3705]=145
Punkte[3706]=105
Punkte[3707]=3
Punkte[3708]=82
Punkte[3709]=170
Punkte[3710]=77
Punkte[3711]=134
Punkte[3712]=8
Punkte[3713]=101
Punkte[3714]=14
Punkte[3715]=90
Punkte[3716]=24
Punkte[3717]=125
Punkte[3718]=33
Punkte[3719]=144
Punkte[3720]=12
Punkte[3721]=99
Punkte[3722]=177
Punkte[3723]=93
Punkte[3724]=36
Punkte[3725]=139
Punkte[3726]=41
Punkte[3727]=140
Punkte[3728]=55
Punkte[3729]=111
Punkte[3730]=31
Punkte[3731]=148
Punkte[3732]=92
Punkte[3733]=0
Punkte[3734]=83
Punkte[3735]=178
Punkte[3736]=34
Punkte[3737]=155
Punkte[3738]=67
Punkte[3739]=1
Punkte[3740]=89
Punkte[3741]=18
Punkte[3742]=103
Punkte[3743]=2
Punkte[3744]=72
Punkte[3745]=138
Punkte[3746]=85
Punkte[3747]=20
Punkte[3748]=117
Punkte[3749]=27
Punkte[3750]=159
Punkte[3751]=28
Punkte[3752]=126
Punkte[3753]=7
Punkte[3754]=145
Punkte[3755]=86
Punkte[3756]=129
Punkte[3757]=0
Punkte[3758]=73
Punkte[3759]=175
Punkte[3760]=64
Punkte[3761]=151
Punkte[3762]=18
Punkte[3763]=92
Punkte[3764]=10
Punkte[3765]=115
Punkte[3766]=56
Punkte[3767]=168
Punkte[3768]=88
Punkte[3769]=141
Punkte[3770]=69
Punkte[3771]=149
Punkte[3772]=76
Punkte[3773]=154
Punkte[3774]=19
Punkte[3775]=116
Punkte[3776]=48
Punkte[3777]=79
Punkte[3778]=14
Punkte[3779]=85
Punkte[3780]=7
Punkte[3781]=86
Punkte[3782]=137
Punkte[3783]=66
Punkte[3784]=163
Punkte[3785]=52
Punkte[3786]=142
Punkte[3787]=72
Punkte[3788]=155
Punkte[3789]=17
Punkte[3790]=117
Punkte[3791]=28
Punkte[3792]=110
Punkte[3793]=24
Punkte[3794]=101
Punkte[3795]=36
Punkte[3796]=146
Punkte[3797]=70
Punkte[3798]=167
Punkte[3799]=102
Punkte[3800]=23
Punkte[3801]=106
Punkte[3802]=0
Punkte[3803]=125
Punkte[3804]=50
Punkte[3805]=137
Punkte[3806]=27
Punkte[3807]=132
Punkte[3808]=21
Punkte[3809]=97
Punkte[3810]=10
Punkte[3811]=107
Punkte[3812]=38
Punkte[3813]=104
Punkte[3814]=7
Punkte[3815]=112
Punkte[3816]=15
Punkte[3817]=90
Punkte[3818]=25
Punkte[3819]=133
Punkte[3820]=74
Punkte[3821]=136
Punkte[3822]=18
Punkte[3823]=80
Punkte[3824]=13
Punkte[3825]=83
Punkte[3826]=138
Punkte[3827]=100
Punkte[3828]=22
Punkte[3829]=143
Punkte[3830]=59
Punkte[3831]=113
Punkte[3832]=40
Punkte[3833]=128
Punkte[3834]=12
Punkte[3835]=146
Punkte[3836]=24
Punkte[3837]=152
Punkte[3838]=77
Punkte[3839]=121
Punkte[3840]=21
Punkte[3841]=94
Punkte[3842]=164
Punkte[3843]=47
Punkte[3844]=107
Punkte[3845]=173
Punkte[3846]=116
Punkte[3847]=175
Punkte[3848]=76
Punkte[3849]=163
Punkte[3850]=89
Punkte[3851]=135
Punkte[3852]=49
Punkte[3853]=147
Punkte[3854]=72
Punkte[3855]=176
Punkte[3856]=105
Punkte[3857]=28
Punkte[3858]=153
Punkte[3859]=31
Punkte[3860]=130
Punkte[3861]=57
Punkte[3862]=115
Punkte[3863]=67
Punkte[3864]=2
Punkte[3865]=75
Punkte[3866]=0
Punkte[3867]=37
Punkte[3868]=144
Punkte[3869]=71
Punkte[3870]=121
Punkte[3871]=52
Punkte[3872]=132
Punkte[3873]=170
Punkte[3874]=106
Punkte[3875]=6
Punkte[3876]=107
Punkte[3877]=7
Punkte[3878]=91
Punkte[3879]=16
Punkte[3880]=142
Punkte[3881]=74
Punkte[3882]=171
Punkte[3883]=104
Punkte[3884]=46
Punkte[3885]=143
Punkte[3886]=39
Punkte[3887]=128
Punkte[3888]=33
Punkte[3889]=139
Punkte[3890]=84
Punkte[3891]=157
Punkte[3892]=53
Punkte[3893]=127
Punkte[3894]=36
Punkte[3895]=129
Punkte[3896]=2
Punkte[3897]=94
Punkte[3898]=28
Punkte[3899]=118
Punkte[3900]=10
Punkte[3901]=44
Punkte[3902]=145
Punkte[3903]=59
Punkte[3904]=134
Punkte[3905]=5
Punkte[3906]=119
Punkte[3907]=43
Punkte[3908]=141
Punkte[3909]=91
Punkte[3910]=177
Punkte[3911]=58
Punkte[3912]=153
Punkte[3913]=78
Punkte[3914]=9
Punkte[3915]=70
Punkte[3916]=173
Punkte[3917]=89
Punkte[3918]=159
Punkte[3919]=83
Punkte[3920]=162
Punkte[3921]=45
Punkte[3922]=98
Punkte[3923]=7
Punkte[3924]=94
Punkte[3925]=166
Punkte[3926]=80
Punkte[3927]=147
Punkte[3928]=18
Punkte[3929]=110
Punkte[3930]=15
Punkte[3931]=148
Punkte[3932]=17
Punkte[3933]=102
Punkte[3934]=14
Punkte[3935]=90
Punkte[3936]=136
Punkte[3937]=30
Punkte[3938]=141
Punkte[3939]=66
Punkte[3940]=145
Punkte[3941]=68
Punkte[3942]=169
Punkte[3943]=96
Punkte[3944]=12
Punkte[3945]=122
Punkte[3946]=13
Punkte[3947]=98
Punkte[3948]=153
Punkte[3949]=42
Punkte[3950]=118
Punkte[3951]=178
Punkte[3952]=121
Punkte[3953]=65
Punkte[3954]=166
Punkte[3955]=103
Punkte[3956]=24
Punkte[3957]=156
Punkte[3958]=91
Punkte[3959]=150
Punkte[3960]=40
Punkte[3961]=131
Punkte[3962]=61
Punkte[3963]=146
Punkte[3964]=39
Punkte[3965]=167
Punkte[3966]=73
Punkte[3967]=161
Punkte[3968]=88
Punkte[3969]=15
Punkte[3970]=122
Punkte[3971]=22
Punkte[3972]=119
Punkte[3973]=71
Punkte[3974]=172
Punkte[3975]=75
Punkte[3976]=152
Punkte[3977]=25
Punkte[3978]=109
Punkte[3979]=12
Punkte[3980]=149
Punkte[3981]=91
Punkte[3982]=175
Punkte[3983]=74
Punkte[3984]=143
Punkte[3985]=77
Punkte[3986]=126
Punkte[3987]=9
Punkte[3988]=84
Punkte[3989]=39
Punkte[3990]=141
Punkte[3991]=38
Punkte[3992]=154
Punkte[3993]=121
Punkte[3994]=5
Punkte[3995]=94
Punkte[3996]=31
Punkte[3997]=163
Punkte[3998]=73
Punkte[3999]=136
Punkte[4000]=79
Punkte[4001]=46


;ENDFOLD (USER EXT)
;ENDFOLD (EXTERNAL DECLARATIONS)
DECL E6POS KM_1={X 270.508820,Y 129.418152,Z 50.0000,A 0.0,B -180.000,C 0.0,S 6,T 26,E1 0.0,E2 0.0,E3 0.0,E4 0.0,E5 0.0,E6 0.0}
ENDDAT
